# B&R Automation Studio project MotionProyect
Automation Studio 4.11.2.75; Proyecto para realizar las practicas realizada para el curso de motion 27-11-24; technology packages: Acp10Arnc0 5.15.1

## Configuration Demo

CPU 4PPC70.0702-23B, AutomationRuntime F4.92, Build 4.1.2, Safety 0.0, Vc V4.72.5

### Task classes (Cpu.sw)
```
Cyclic#4:
  AxisProgra <- Source.AxisProgram.prg
Libraries: McBase, CoTrace, AsZip, FileIO, runtime, MpAxis, McAxis, MpBase, McAcpAx
```

### Hardware
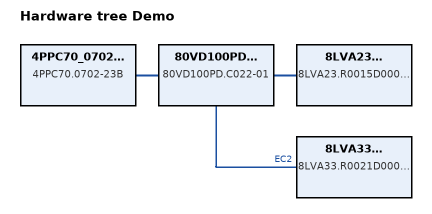
```
4PPC70_0702_23B : 4PPC70.0702-23B v1.5.4.0
  Connector IF2:
    ActivateDevice = 1
    Mode = Manual
    InternetAddress = 192.168.150.95
    SubnetMask = 255.255.255.0
    ActivateSnmp = 2
  ConfigurationID = mappMotion_Demo
  FileDevice1
  FileDeviceName1 = USER
  FileDevicePath1 = USER_PATH
  ActivateOpcUa = 1
  OpcUaInformationModels_PV_Version = 1
  KeyMappingFile = VC\4PPC70_0702_23B.dis
80VD100PD.C022-01 : 80VD100PD.C022-01 v2.5.0.0  [PLK1 -> 4PPC70_0702_23B.IF1 (NodeNumber=2) [Cable Type=PowerlinkCable, Length=10, Version=1.0.0.3]; EC1 -> 8LVA23.R0015D000-0.EC; EC2 -> 8LVA33.R0021D000-0.EC; MT2 -> 8LVA33.R0021D000-0.MT]
  DriveConfiguration/Module:
    McAcoposTypeID = AcoposMicroDConfig
    ActivateACOPOSSimulationOnPLC = 0
  DriveConfiguration/Encoder/EncoderX6A/InterfaceType:
    ResolverPolepairs = 1
  DriveConfiguration/Encoder/EncoderX6B/InterfaceType:
    ResolverPolepairs = 1
  DriveConfiguration/Channel[1]/RealAxis:
    AxisReference = gAxis_1
    MechanicalElementsIsInvisible = 0
  DriveConfiguration/Channel[1]/RealAxis/MechanicalElements/Gearbox:
    InputIsReadOnly = 0
    Input = 1
    OutputIsReadOnly = 0
    Output = 1
  DriveConfiguration/Channel[1]/RealAxis/MechanicalElements/RotaryToLinearTransformation:
    ReferenceDistanceIsReadOnly = 0
    ReferenceDistance = 1
  DriveConfiguration/Channel[1]/RealAxis/Controller:
    ModeIsReadOnly = 0
    Mode = PositionController
  DriveConfiguration/Channel[1]/RealAxis/Controller/Mode/Position:
    ProportionalGain = 50.0
    IntegrationTime = 0.0
    PredictionTime = 0.0004
    TotalDelayTime = 0.0004
  DriveConfiguration/Channel[1]/RealAxis/Controller/Mode/Speed:
    ProportionalGainIsReadOnly = 0
    ProportionalGain = 2.0
    IntegrationTimeIsReadOnly = 0
    IntegrationTime = 0.0
    FilterTimeIsReadOnly = 0
    FilterTime = 0.0
  DriveConfiguration/Channel[1]/RealAxis/Controller/Mode/LoopFilters:
    LoopFilterXIsReadOnly = 0
    LoopFilter1 = NotUsed
    LoopFilter2 = NotUsed
    LoopFilter3 = NotUsed
  DriveConfiguration/Channel[1]/RealAxis/Homing:
    ModeIsReadOnly = 0
    Mode = Direct
  DriveConfiguration/Channel[1]/RealAxis/Homing/Mode:
    Position = 0.0
    ReferencePulse = NotUsed
  DriveConfiguration/Channel[1]/RealAxis/Homing:
    RestorePositionVariable = 
  DriveConfiguration/Channel[1]/RealAxis/StopReaction:
    QuickstopIsReadOnly = 0
    Quickstop = DecelerationLimit
    DriveErrorIsReadOnly = 0
    DriveError = DecelerationLimit
  DriveConfiguration/Channel[1]/RealAxis/MovementErrorLimits:
    PositionError = 1.0
    VelocityErrorMonitoring = Automatic1
  DriveConfiguration/Channel[1]/RealAxis:
    JerkFilterIsReadOnly = 0
    JerkFilter = NotUsed
  DriveConfiguration/Channel[1]/RealAxis/DigitalInputs/HomingSwitch:
    SourceIsReadOnly = 0
    Source = NotUsed
    Level = High
  DriveConfiguration/Channel[1]/RealAxis/DigitalInputs/PositiveLimitSwitch:
    SourceIsReadOnly = 0
    Source = NotUsed
    Level = High
  DriveConfiguration/Channel[1]/RealAxis/DigitalInputs/NegativeLimitSwitch:
    SourceIsReadOnly = 0
    Source = NotUsed
    Level = High
  DriveConfiguration/Channel[1]/RealAxis/DigitalInputs/Trigger1:
    Source = X2Trigger1
    Level = High
  DriveConfiguration/Channel[1]/RealAxis/DigitalInputs/Trigger2:
    Source = X2Trigger2
    Level = High
  DriveConfiguration/Channel[1]/RealAxis/DigitalInputs/Quickstop:
    Input = Trigger2
  DriveConfiguration/Channel[1]/RealAxis/Simulation:
    SimulationModeOnPLC = SetValueGeneration
    SimulationModeOnACOPOS = NotUsed
  DriveConfiguration/Channel[2]/RealAxis:
    AxisReference = gAxis_2
    MechanicalElementsIsInvisible = 0
  DriveConfiguration/Channel[2]/RealAxis/MechanicalElements/Gearbox:
    InputIsReadOnly = 0
    Input = 1
    OutputIsReadOnly = 0
    Output = 1
  DriveConfiguration/Channel[2]/RealAxis/MechanicalElements/RotaryToLinearTransformation:
    ReferenceDistanceIsReadOnly = 0
    ReferenceDistance = 1
  DriveConfiguration/Channel[2]/RealAxis/Controller:
    ModeIsReadOnly = 0
    Mode = PositionController
  DriveConfiguration/Channel[2]/RealAxis/Controller/Mode/Position:
    ProportionalGain = 50.0
    IntegrationTime = 0.0
    PredictionTime = 0.0004
    TotalDelayTime = 0.0004
  DriveConfiguration/Channel[2]/RealAxis/Controller/Mode/Speed:
    ProportionalGainIsReadOnly = 0
    ProportionalGain = 2.0
    IntegrationTimeIsReadOnly = 0
    IntegrationTime = 0.0
    FilterTimeIsReadOnly = 0
    FilterTime = 0.0
  DriveConfiguration/Channel[2]/RealAxis/Controller/Mode/LoopFilters:
    LoopFilterXIsReadOnly = 0
    LoopFilter1 = NotUsed
    LoopFilter2 = NotUsed
    LoopFilter3 = NotUsed
  DriveConfiguration/Channel[2]/RealAxis/Homing:
    ModeIsReadOnly = 0
    Mode = Direct
  DriveConfiguration/Channel[2]/RealAxis/Homing/Mode:
    Position = 0.0
    ReferencePulse = NotUsed
  DriveConfiguration/Channel[2]/RealAxis/Homing:
    RestorePositionVariable = 
  DriveConfiguration/Channel[2]/RealAxis/StopReaction:
    QuickstopIsReadOnly = 0
    Quickstop = DecelerationLimit
    DriveErrorIsReadOnly = 0
    DriveError = DecelerationLimit
  DriveConfiguration/Channel[2]/RealAxis/MovementErrorLimits:
    PositionError = 1.0
    VelocityErrorMonitoring = Automatic1
  DriveConfiguration/Channel[2]/RealAxis:
    JerkFilterIsReadOnly = 0
    JerkFilter = NotUsed
  DriveConfiguration/Channel[2]/RealAxis/DigitalInputs/HomingSwitch:
    SourceIsReadOnly = 0
    Source = NotUsed
    Level = High
  DriveConfiguration/Channel[2]/RealAxis/DigitalInputs/PositiveLimitSwitch:
    SourceIsReadOnly = 0
    Source = NotUsed
    Level = High
  DriveConfiguration/Channel[2]/RealAxis/DigitalInputs/NegativeLimitSwitch:
    SourceIsReadOnly = 0
    Source = NotUsed
    Level = High
  DriveConfiguration/Channel[2]/RealAxis/DigitalInputs/Trigger1:
    Source = X2Trigger1
    Level = High
  DriveConfiguration/Channel[2]/RealAxis/DigitalInputs/Trigger2:
    Source = X2Trigger2
    Level = High
  DriveConfiguration/Channel[2]/RealAxis/DigitalInputs/Quickstop:
    Input = Trigger2
  DriveConfiguration/Channel[2]/RealAxis/Simulation:
    SimulationModeOnPLC = SetValueGeneration
    SimulationModeOnACOPOS = NotUsed
8LVA23.R0015D000-0 : 8LVA23.R0015D000-0 v2.2.0.3  [EC -> 80VD100PD.C022-01.EC1; MT -> 80VD100PD.C022-01.MT1]
  M1/MotorParameters:
    MOTOR_AMB_TEMP_RATED = 40
8LVA33.R0021D000-0 : 8LVA33.R0021D000-0 v2.2.0.3  [EC -> 80VD100PD.C022-01.EC2; MT -> 80VD100PD.C022-01.MT2]
  M1/MotorParameters:
    MOTOR_AMB_TEMP_RATED = 40
```

### IoMap.iom - 4PPC70_0702_23B/IoMap.iom
```iecst
VAR_CONFIG
	::AxisSequence.io.di_PowerMotors AT %IX."4XP0043.00-00W".DigitalInput01;
	::AxisSequence.io.di_StartSequence AT %IX."4XP0043.00-00W".DigitalInput02;
	::AxisSequence.io.di_StopSequence AT %IX."4XP0043.00-00W".DigitalInput03;
END_VAR
```

### Acp10cfg.ncc - 4PPC70_0702_23B/Motion/Acp10cfg.ncc
```
NcConfiguration (Version=5.15.1, NcSwId=Acp10)
  ACP10CF1_typ:
    cnt_nettrc_rec_drive = 1500
    bufsize_trace_upload = 1200
    tc_nc_man_task = Cyclic #1
    glob_pv_as_ncobject = Yes
    ncsys_dl_broadcast = Yes
    ncsys_dl_acp_reset = Yes
    safemc_log_err_to_ax = Yes
    network_init:
      ncsw_init_execute = Yes
      automatic_execute = No
      node_nr_warning = Yes
      net_err_before_ncact = Yes
    nettrc:
      enter_parsecrec = Yes
      enter_ncaction = Yes
      save_ring_startidx = Yes
    cam_prof_download:
      cam_dat_dl_parallel = No
      tc_cam_dl_parallel = Task class for NC Manager task
    plk_if[0]:
      if_name = IF1
      tc_CycDat_PLCopen = Task class for NC Manager task
      mc_broadcast_extdat = No
```

### Acp10map.ncm - 4PPC70_0702_23B/Motion/Acp10map.ncm
```
NcMapping (NcSwId=Acp10, DisabledNodesAreHidden=False)
  NcObject gAxis02 (ModuleId=80VD100PD.C022-01, Type=ncAXIS, Channel=2, AcoposSimulation=Off, InitParameter=gAxis02i, AcoposParameter=gAxis02a, AdditionalData=PLCopen_ModPos="36000,100" , Disabled=FALSE, ModuleDisabled=FALSE)
  NcObject gAxis01 (ModuleId=80VD100PD.C022-01, Type=ncAXIS, Channel=1, AcoposSimulation=Off, InitParameter=gAxis01i, AcoposParameter=gAxis01a, AdditionalData=PLCopen_ModPos="36000,100" , Disabled=FALSE, ModuleDisabled=FALSE)
  NcObject 80VD100PD.C022-01_ncV_AXIS2 (ModuleId=80VD100PD.C022-01, Type=ncV_AXIS, Channel=2, Disabled=TRUE, ModuleDisabled=FALSE)
  NcObject 80VD100PD.C022-01_ncV_AXIS1 (ModuleId=80VD100PD.C022-01, Type=ncV_AXIS, Channel=1, Disabled=TRUE, ModuleDisabled=FALSE)
```

### Axis1.axis - 4PPC70_0702_23B/mappMotion/Axis1.axis
```
Element gAxis_1 (Type=axis)
  BaseTypeIsReadOnly = 0
  BaseType = RotaryPeriodic
    MeasurementUnitIsReadOnly = 0
    MeasurementUnit = 17476
    MeasurementResolutionIsReadOnly = 0
    MeasurementResolution = 0.01
    CountDirectionIsReadOnly = 0
    CountDirection = Standard
    PeriodSettings:
      Period = 360.0
  MovementLimitsIsReadOnly = 0
  MovementLimits = Internal
    Position:
      LowerLimitMin = -1.79769313486231E308
      UpperLimitMax = 1.79769313486231E308
      LowerLimit = -1000.0
      UpperLimit = 1000.0
    VelocityIsReadOnly = 0
    Velocity:
      VelocityMax = 3.4E38
      Velocity = 1000
    AccelerationIsReadOnly = 0
    Acceleration:
      AccelerationMax = 3.4E38
      Acceleration = 1000
    DecelerationIsReadOnly = 0
    Deceleration:
      DecelerationMax = 3.4E38
      Deceleration = 1000
  Alarms = None
```

### Axis2.axis - 4PPC70_0702_23B/mappMotion/Axis2.axis
```
Element gAxis_2 (Type=axis)
  BaseTypeIsReadOnly = 0
  BaseType = RotaryPeriodic
    MeasurementUnitIsReadOnly = 0
    MeasurementUnit = 17476
    MeasurementResolutionIsReadOnly = 0
    MeasurementResolution = 0.01
    CountDirectionIsReadOnly = 0
    CountDirection = Standard
    PeriodSettings:
      Period = 360.0
  MovementLimitsIsReadOnly = 0
  MovementLimits = Internal
    Position:
      LowerLimitMin = -1.79769313486231E308
      UpperLimitMax = 1.79769313486231E308
      LowerLimit = -1000.0
      UpperLimit = 1000.0
    VelocityIsReadOnly = 0
    Velocity:
      VelocityMax = 3.4E38
      Velocity = 1400
    AccelerationIsReadOnly = 0
    Acceleration:
      AccelerationMax = 3.4E38
      Acceleration = 1000
    DecelerationIsReadOnly = 0
    Deceleration:
      DecelerationMax = 3.4E38
      Deceleration = 1000
  Alarms = None
```

### CfgAutomat.axisfeature - 4PPC70_0702_23B/mappMotion/CfgAutomat.axisfeature
```
Element Feature_1 (Type=axisfeature)
  Type = CamAutomat
    CamAutomatType = ACOPOS
      CommonParameters:
        Master:
          ValueSource = SetPosition
            AxisReference = gAxis_1
            MaxVelocity = 30
          StartPosition = 0.0
          StartInterval = MasterAxisPeriod
        AdvancedParameters:
          StartStateParameters:
            StartState = 0
            RelMasterStartPos = 0.0
          AdditiveAxes:
            AdditiveMasterValueSource = NotUsed
            AdditiveSlaveValueSource = NotUsed
          MasterStartPositionMode = NotEvaluatedAnew
          ControlSettings:
            CrossLeftBoundary = PositionLimitedHorizontal
            CamChangeImmediately = CurrentMasterMoveDir
          MessageSettings:
            ErrorsInStandby = NoErrorMessages
          TriggerAndLatch:
            Trigger1Delay = 0.0
            Trigger2Delay = 0.0
            SlaveLatchParID = 0
          EventParIDs
          StartIntervals
          Factors:
            SlaveFactorParID = 0
      States:
        State0 = Used
          Events:
            Event[0]:
              Type = StateEnd
              Transition = Immediately
              SynchronousUpdate = NotUsed
              NextState = 1
        State[1]:
          Cam = Predefined
            PredefinedCam = OneToOne
          MasterFactor = 600
          SlaveFactor = 0
          CompensationMode = NoCompensation
          AdvancedParameters:
            RepeatCounterInit = 0
            MasterValueSource = CommonMaster
          Events:
            Event[0]:
              Type = Signal1FromPLC
              Transition = EndOfState
              SynchronousUpdate = NotUsed
              NextState = 2
            Event[1]:
              Type = StateEnd
              Transition = Immediately
              SynchronousUpdate = NotUsed
              NextState = 1
        State[2]:
          Cam = Predefined
            PredefinedCam = ZeroPoint
          MasterFactor = 1
          SlaveFactor = 1
          CompensationMode = DistancesBetweenCams
            MasterDistance = 20
            SlaveDistance = 170
            AdvancedParameters = NotUsed
          AdvancedParameters:
            RepeatCounterInit = 0
            MasterValueSource = CommonMaster
          Events:
            Event[0]:
              Type = StateEnd
              Transition = EndOfState
              SynchronousUpdate = NotUsed
              NextState = 3
        State[3]:
          Cam = Predefined
            PredefinedCam = OneToOne
          MasterFactor = 400
          SlaveFactor = 100
          CompensationMode = NoCompensation
          AdvancedParameters:
            RepeatCounterInit = 0
            MasterValueSource = CommonMaster
          Events:
            Event[0]:
              Type = StateEnd
              Transition = EndOfState
              SynchronousUpdate = NotUsed
              NextState = 4
        State[4]:
          Cam = Predefined
            PredefinedCam = ZeroPoint
          MasterFactor = 1
          SlaveFactor = 1
          CompensationMode = DistancesBetweenCams
            MasterDistance = 20
            SlaveDistance = 180
            AdvancedParameters = NotUsed
          AdvancedParameters:
            RepeatCounterInit = 0
            MasterValueSource = CommonMaster
          Events:
            Event[0]:
              Type = StateEnd
              Transition = EndOfState
              SynchronousUpdate = NotUsed
              NextState = 1
            Event[1]:
              Type = Signal1FromPLC
              Transition = EndOfState
              SynchronousUpdate = NotUsed
              NextState = 2
```

## Logical view

Binary libraries used (declarations not repeated): operator, runtime, astime, AsIecCon, McBase 5.20.2, CoTrace, AsZip, FileIO, MpAxis 5.20.2, McAxis 5.20.2, MpBase, McAcpAx 5.20.2

### Global.typ - Global data types
```iecst
TYPE
	AxisSequence_typ : 	STRUCT
		cmd : AxisSequence_cmd_typ;
		status : AxisSequence_status_typ;
		io : AxisSequence_io_typ;
		state : AxisSequence_enum;
		couplingParam : MpAxisCouplingParType;
		camSequencer : USINT;
		parameters : ARRAY[1..MAX_AXIS]OF MpAxisBasicParType;
	END_STRUCT;
	AxisSequence_cmd_typ : 	STRUCT
		AutoTune : ARRAY[1..MAX_AXIS]OF BOOL;
		Enable : ARRAY[1..MAX_AXIS]OF BOOL;
		ErrorReset : ARRAY[1..MAX_AXIS]OF BOOL;
		Update : ARRAY[1..MAX_AXIS]OF BOOL;
		Power : ARRAY[1..MAX_AXIS]OF BOOL;
		Home : ARRAY[1..MAX_AXIS]OF BOOL;
		MoveVelocity : ARRAY[1..MAX_AXIS]OF BOOL;
		MoveAbsolute : ARRAY[1..MAX_AXIS]OF BOOL;
		MoveAdditive : ARRAY[1..MAX_AXIS]OF BOOL;
		Stop : ARRAY[1..MAX_AXIS]OF BOOL;
		JogPositive : ARRAY[1..MAX_AXIS]OF BOOL;
		JogNegative : ARRAY[1..MAX_AXIS]OF BOOL;
	END_STRUCT;
	AxisSequence_status_typ : 	STRUCT
		PowerMotors : BOOL;
		StartSequence : BOOL;
		StopSequence : BOOL;
		Active : ARRAY[1..MAX_AXIS]OF BOOL;
		Error : ARRAY[1..MAX_AXIS]OF BOOL;
		StatusID : ARRAY[1..MAX_AXIS]OF DINT;
		UpdateDone : ARRAY[1..MAX_AXIS]OF BOOL;
		Position : ARRAY[1..MAX_AXIS]OF LREAL;
		Velocity : ARRAY[1..MAX_AXIS]OF REAL;
		CommandBusy : ARRAY[1..MAX_AXIS]OF BOOL;
		CommandAborted : ARRAY[1..MAX_AXIS]OF BOOL;
		PowerOn : ARRAY[1..MAX_AXIS]OF BOOL;
		IsHomed : ARRAY[1..MAX_AXIS]OF BOOL;
		InVelocity : ARRAY[1..MAX_AXIS]OF BOOL;
		InPosition : ARRAY[1..MAX_AXIS]OF BOOL;
		MoveActive : ARRAY[1..MAX_AXIS]OF BOOL;
		MoveDone : ARRAY[1..MAX_AXIS]OF BOOL;
		Info : ARRAY[1..MAX_AXIS]OF MpAxisBasicInfoType;
	END_STRUCT;
	AxisSequence_io_typ : 	STRUCT
		di_PowerMotors : BOOL;
		di_StartSequence : BOOL;
		di_StopSequence : BOOL;
	END_STRUCT;
	AxisSequence_enum :
		(
		DISABLED := 0,
		WAIT := 5,
		STEP_1 := 10,
		STEP_2 := 20,
		STEP_3 := 30,
		STEP_4 := 40,
		STEP_5 := 50,
		STEP_6 := 60,
		STEP_7 := 70,
		STEP_8 := 80,
		ERROR := 100
		);
END_TYPE
```

### Constans.var
```iecst
VAR CONSTANT
	MAX_AXIS : USINT := 2;
END_VAR
```

### Global.var - Global variables
```iecst
VAR
	MpAxisBasic_0 : ARRAY[1..MAX_AXIS] OF MpAxisBasic;
	AxisParameters : ARRAY[1..MAX_AXIS] OF MpAxisBasicParType;
	AxisInfo : ARRAY[1..MAX_AXIS] OF MpAxisBasicInfoType;
END_VAR
```


### Program Logical/Source/AxisProgram (IEC)

#### Main.st - Init, cyclic, exit code
```iecst
PROGRAM _INIT
	(* INIT AXIS *)
	FOR i:= 1 TO MAX_AXIS DO

		MpAxisBasic_0[i].Enable	:= TRUE;

		AxisParameters[i].Position		:= 100;
		AxisParameters[i].Velocity		:= 10.0;
		AxisParameters[i].Acceleration	:= 50.0;
		AxisParameters[i].Deceleration	:= 50.0;

	END_FOR;

END_PROGRAM

PROGRAM _CYCLIC

	(* CYCLIC AXIS *)
	MpAxisBasic_0[1].MpLink		:= ADR(gAxis_1);
	MpAxisBasic_0[1].Parameters	:= ADR(AxisParameters[1]);
	AxisInfo[1]					:= MpAxisBasic_0[1].Info;
	MpAxisBasic_0[1]();

	MpAxisBasic_0[2].MpLink		:= ADR(gAxis_2);
	MpAxisBasic_0[2].Parameters	:= ADR(AxisParameters[2]);
	AxisInfo[2]					:= MpAxisBasic_0[2].Info;
	MpAxisBasic_0[2]();

END_PROGRAM

PROGRAM _EXIT

	(* EXIT AXIS *)
	FOR i:= 1 TO MAX_AXIS DO
		MpAxisBasic_0[1].Enable	:= FALSE;
	END_FOR;

END_PROGRAM
```

#### Types.typ - Local data types
```iecst
TYPE
	AxisSequence_typ : 	STRUCT
		cmd : AxisSequence_cmd_typ;
		status : AxisSequence_status_typ;
		io : AxisSequence_io_typ;
		state : AxisSequence_enum;
	END_STRUCT;
	AxisSequence_cmd_typ : 	STRUCT
		Enable : ARRAY[1..MAX_AXIS]OF BOOL;
		ErrorReset : ARRAY[1..MAX_AXIS]OF BOOL;
		Update : ARRAY[1..MAX_AXIS]OF BOOL;
		Power : ARRAY[1..MAX_AXIS]OF BOOL;
		Home : ARRAY[1..MAX_AXIS]OF BOOL;
		MoveVelocity : ARRAY[1..MAX_AXIS]OF BOOL;
		MoveAbsolute : ARRAY[1..MAX_AXIS]OF BOOL;
		Stop : ARRAY[1..MAX_AXIS]OF BOOL;
		JogPositive : ARRAY[1..MAX_AXIS]OF BOOL;
		JogNegative : ARRAY[1..MAX_AXIS]OF BOOL;
	END_STRUCT;
	AxisSequence_status_typ : 	STRUCT
		PowerMotors : BOOL;
		StartSequence : BOOL;
		StopSequence : BOOL;
		Active : ARRAY[1..MAX_AXIS]OF BOOL;
		Error : ARRAY[1..MAX_AXIS]OF BOOL;
		StatusID : ARRAY[1..MAX_AXIS]OF BOOL;
		UpdateDone : ARRAY[1..MAX_AXIS]OF BOOL;
		Position : ARRAY[1..MAX_AXIS]OF BOOL;
		Velocity : ARRAY[1..MAX_AXIS]OF BOOL;
		CommandBusy : ARRAY[1..MAX_AXIS]OF BOOL;
		CommandAborted : ARRAY[1..MAX_AXIS]OF BOOL;
		PowerOn : ARRAY[1..MAX_AXIS]OF BOOL;
		IsHomed : ARRAY[1..MAX_AXIS]OF BOOL;
		InVelocity : ARRAY[1..MAX_AXIS]OF BOOL;
		InPosition : ARRAY[1..MAX_AXIS]OF BOOL;
		MoveActive : ARRAY[1..MAX_AXIS]OF BOOL;
		MoveDone : ARRAY[1..MAX_AXIS]OF BOOL;
	END_STRUCT;
	AxisSequence_io_typ : 	STRUCT
	END_STRUCT;
	AxisSequence_enum :
		(
		WAIT := 0,
		STEP_1 := 10,
		STEP_2 := 20,
		STEP_3 := 30,
		STEP_4 := 40,
		STEP_5 := 50,
		STEP_6 := 60,
		STEP_7 := 70,
		STEP_8 := 80,
		ERROR := 100
		);
END_TYPE
```

#### Variables.var
```iecst
VAR
	AxisSequence : AxisSequence_typ;
	i : USINT;
END_VAR
```

#### Sequences.st
```iecst
ACTION AutoSequence180Action:

END_ACTION
```

### Program Logical/Source/AxisCtrl (IEC)

#### Main.st - Init, cyclic, exit code
```iecst
PROGRAM _INIT
	(* INIT AXIS *)
	FOR i:= 1 TO MAX_AXIS DO

		MpAxisBasic_0[i].Enable	:= TRUE;

		AxisSequence.parameters[i].Position		:= 100;
		AxisSequence.parameters[i].Velocity		:= 10.0;
		AxisSequence.parameters[i].Acceleration	:= 50.0;
		AxisSequence.parameters[i].Deceleration	:= 50.0;

	END_FOR;
	(* CYCLIC AXIS *)
	MpAxisBasic_0[1].MpLink		:= ADR(gAxis_1);
	MpAxisBasic_0[1].Parameters	:= ADR(AxisSequence.parameters[1]);
	MpAxisBasic_0[1]();

	MpAxisBasic_0[2].MpLink		:= ADR(gAxis_2);
	MpAxisBasic_0[2].Parameters	:= ADR(AxisSequence.parameters[2]);
	MpAxisBasic_0[2]();

//	AxisSequence.couplingParam.Gear.RatioDenominator 	:= 3600;
//	AxisSequence.couplingParam.Gear.RatioNumerator		:= -3600;
//	MpAxisCoupling_0.MpLinkMaster	:= ADR(gAxis_1);
//	MpAxisCoupling_0.MpLink 		:= ADR(gAxis_2);
//	MpAxisCoupling_0.Parameters		:= ADR(AxisSequence.couplingParam);
	//	MpAxisCoupling_0.Enable			:= TRUE;

	MpAxisCamSequencer_0.MpLinkMaster 	:= ADR(gAxis_1);
	MpAxisCamSequencer_0.MpLink			:= ADR(gAxis_2);
	MpAxisCamSequencer_0.Parameters		:= ADR(CamSequencerParam);
	MpAxisCamSequencer_0.Enable 		:= TRUE;
	CamSequencerParam.CamSequence.Data.DataAddress	:= ADR (CamAutomatParam);
	MpAxisCamSequencer_0();

END_PROGRAM

PROGRAM _CYCLIC
	MpAxisCamSequencer_0.Signal1		:= AxisSequence.io.di_PowerMotors;
	IF EnableSequence THEN
		TapSequencerAction;
	END_IF;

	MpAxisBasic_0[1]();
	MpAxisBasic_0[2]();

	MpAxisCamSequencer_0();
	//MpAxisCoupling_0();
	(* Axis actions *)
	//AxisCtrlCmdAction;

//	/////////// PHYSICAL INPUTS ///////////
//	AxisSequence.status.PowerMotors		:= AxisSequence.io.di_PowerMotors;
//	AxisSequence.status.StartSequence	:= AxisSequence.io.di_StartSequence;
//	AxisSequence.status.StopSequence	:= AxisSequence.io.di_StopSequence;
//
//
//
//	//Timer poweroff condition
//	TON_TurnOffMotors.PT	:= T#2s;
//
//	IF (AxisSequence.status.StopSequence)  THEN
//		TON_TurnOffMotors.IN	:= TRUE;
//	ELSE
//		TON_TurnOffMotors.IN := FALSE;
//	END_IF;
//
//
//
//	FOR i:= 1 TO MAX_AXIS DO
//
//		IF (AxisSequence.state <> STEP_4) AND NOT (AxisSequence.state = STEP_1) THEN
//			AxisSequence.parameters[i].Distance		:= 180;
//			AxisSequence.parameters[i].Velocity		:= 100;
//			AxisSequence.parameters[i].Acceleration := 1000;
//			AxisSequence.parameters[i].Deceleration := 1000;
//			AxisSequence.parameters[i].Direction := mcDIR_POSITIVE;
//		ELSIF (AxisSequence.state = STEP_4) THEN
//			AxisSequence.parameters[i].Distance		:= -540;
//			AxisSequence.parameters[i].Velocity		:= 100;
//			AxisSequence.parameters[i].Acceleration := 1000;
//			AxisSequence.parameters[i].Deceleration := 1000;
//			AxisSequence.parameters[i].Direction 	:= mcDIR_NEGATIVE;
//
//		END_IF;
//
//		//PowerOn condition
//		IF EDGEPOS(AxisSequence.status.PowerMotors)  THEN
//			MpAxisBasic_0[1].Power	:= TRUE;
//			MpAxisBasic_0[2].Power	:= TRUE;
//		END_IF;
//
//		//Stop condition
//		IF AxisSequence.status.StopSequence OR ResetSequence THEN
//			MpAxisBasic_0[i].Home			:= FALSE;
//			MpAxisBasic_0[i].MoveAbsolute	:= FALSE;
//			MpAxisBasic_0[i].MoveAdditive	:= FALSE;
//			MpAxisBasic_0[i].MoveVelocity	:= FALSE;
//			ResetSequence	:= FALSE;
//			//MpAxisBasic_0[i].Stop			:= TRUE;
//			AxisSequence.state	 			:= STEP_1;
//		ELSE
//			//MpAxisBasic_0[i].Stop 		:= FALSE;
//			MpAxisBasic_0[i].ErrorReset	:= FALSE;
//		END_IF;
//
//		//PowerOff condition
//		IF TON_TurnOffMotors.Q  	THEN
//			MpAxisBasic_0[i].Power			:= FALSE;
//			MpAxisBasic_0[i].Home			:= FALSE;
//			MpAxisBasic_0[i].MoveAbsolute	:= FALSE;
//			MpAxisBasic_0[i].MoveAdditive	:= FALSE;
//			MpAxisBasic_0[i].MoveVelocity	:= FALSE;
//			MpAxisBasic_0[i].Stop			:= TRUE;
//			MpAxisBasic_0[i].ErrorReset		:= TRUE;
//			ResetSequence	:= FALSE;
//			AxisSequence.state	 			:= WAIT;
//		END_IF;
//
//
//		//Error condition
//		IF 	MpAxisBasic_0[i].Error THEN
//			AxisSequence.state	:= ERROR;
//		END_IF;
//
//
//
//
//		CASE AxisSequence.state OF
//
//			DISABLED:
//
//				IF 	MpAxisBasic_0[1].Info.ReadyToPowerOn AND (MpAxisBasic_0[2].Info.ReadyToPowerOn) THEN
//					AxisSequence.state	:= WAIT;
//				ELSE
//
//				END_IF;
//
//			WAIT:
//
//				MpAxisBasic_0[i].Stop:= FALSE;
//
//				IF	MpAxisBasic_0[i].Power AND MpAxisBasic_0[i].PowerOn THEN
//					AxisSequence.state	:= STEP_1;
//				END_IF;
//
//			STEP_1:
//
//
//
//				IF (AxisSequence.status.StartSequence) AND (OldStartSequence <> AxisSequence.status.StartSequence) THEN
//					AxisSequence.parameters[1].Homing.Position 	:= 30;
//					AxisSequence.parameters[2].Homing.Position	:= 200;
//					AxisSequence.parameters[1].Homing.Mode 	:= mcHOMING_DIRECT ;
//					AxisSequence.parameters[2].Homing.Mode 	:= mcHOMING_DIRECT ;
//					MpAxisBasic_0[1].Home	:= TRUE;
//					MpAxisBasic_0[2].Home	:= TRUE;
//					PermissionToHome		:= TRUE;
//				END_IF;
//
//				IF (MpAxisBasic_0[1].IsHomed AND MpAxisBasic_0[2].IsHomed) AND (MpAxisBasic_0[1].Position = 30)
//					AND MpAxisBasic_0[2].Position = 200 AND PermissionToHome AND (CountSequence = 0) THEN
//
//					MpAxisBasic_0[1].Home	:= FALSE;
//					MpAxisBasic_0[2].Home	:= FALSE;
//					PermissionToHome		:= FALSE;
//					PermissionToStart		:= TRUE;
//
//				END_IF;
//
//				IF PermissionToStart THEN
//					AxisSequence.parameters[1].Position	:= 0;
//					AxisSequence.parameters[2].Position	:= 0;
//					AxisSequence.parameters[1].Direction := mcDIR_SHORTEST_WAY;
//					AxisSequence.parameters[2].Direction := mcDIR_SHORTEST_WAY;
//
//					MpAxisBasic_0[1].MoveAbsolute	:= TRUE;
//					MpAxisBasic_0[2].MoveAbsolute	:= TRUE;
//				END_IF;
//
//				IF MpAxisBasic_0[1].InPosition AND MpAxisBasic_0[1].MoveDone THEN
//					MpAxisBasic_0[1].MoveAbsolute	:= FALSE;
//					FinishSequence[1]				:= TRUE;
//				END_IF;
//
//				IF MpAxisBasic_0[2].InPosition AND MpAxisBasic_0[2].MoveDone THEN
//					MpAxisBasic_0[2].MoveAbsolute	:= FALSE;
//					FinishSequence[2]				:= TRUE;
//				END_IF;
//
//				IF FinishSequence[1] AND FinishSequence[2] THEN
//					FinishSequence[1]		:= FALSE;
//					FinishSequence[2]		:= FALSE;
//					PermissionToStart		:= FALSE;
//					CountSequence			:= 1;
//					AxisSequence.state		:= STEP_2;
//				END_IF;
//
//			STEP_2: //+180° Axis 1
//
//				IF (CountSequence <7) THEN
//					MpAxisBasic_0[1].MoveAdditive	:= TRUE;
//					IF MpAxisBasic_0[1].InPosition AND (MpAxisBasic_0[1].MoveDone) THEN
//						MpAxisBasic_0[1].MoveAdditive	:= FALSE;
//						CountSequence 					:= CountSequence + 1;
//						AxisSequence.state				:= STEP_3;
//					END_IF;
//				END_IF;
//
//				IF (CountSequence = 7) THEN
//					AxisSequence.state	:= STEP_4;
//				END_IF;
//
//			STEP_3: //+180 Axis 2
//
//				IF (CountSequence <7) THEN
//					MpAxisBasic_0[2].MoveAdditive := TRUE;
//					IF MpAxisBasic_0[2].InPosition AND (MpAxisBasic_0[2].MoveDone) THEN
//						MpAxisBasic_0[2].MoveAdditive	:= FALSE;
//						CountSequence 					:= CountSequence + 1;
//						AxisSequence.state				:= STEP_2;
//					END_IF;
//				END_IF;
//
//			STEP_4:
//
//				MpAxisBasic_0[i].MoveAdditive := TRUE;
//
//				IF MpAxisBasic_0[1].InPosition AND MpAxisBasic_0[1].MoveDone THEN
//					MpAxisBasic_0[1].MoveAdditive	:= FALSE;
//					FinishSequence[1]				:= TRUE;
//				END_IF;
//
//				IF MpAxisBasic_0[2].InPosition AND MpAxisBasic_0[2].MoveDone THEN
//					MpAxisBasic_0[2].MoveAdditive	:= FALSE;
//					FinishSequence[2]				:= TRUE;
//				END_IF;
//
//				IF FinishSequence[1] AND FinishSequence[2] THEN
//					FinishSequence[1]		:= FALSE;
//					FinishSequence[2]		:= FALSE;
//					ResetSequence			:= TRUE;
//					CountSequence			:= 0;
//					AxisSequence.state		:= STEP_1;
//				END_IF;
//
//
//			ERROR:
//
//				MpAxisBasic_0[i].MoveAdditive	:= FALSE;
//				IF NOT(MpAxisBasic_0[1].Error) AND NOT(MpAxisBasic_0[2].Error)THEN
//					AxisSequence.state	:= WAIT;
//				END_IF;
//
//
//		END_CASE;
//
//
//		MpAxisBasic_0[i]();
//	END_FOR;
//
//
//	//Old variables
//	OldStartSequence := AxisSequence.status.StartSequence;
//
//	//Call Functions blocks
//	//AxisCtrlStatusAction;
//	TON_TurnOffMotors();
//

END_PROGRAM

PROGRAM _EXIT

	(* EXIT AXIS *)
	FOR i:= 1 TO MAX_AXIS DO
		MpAxisBasic_0[i].Enable	:= FALSE;
	END_FOR;

END_PROGRAM
```

#### Variables.var
```iecst
VAR
	MpAxisBasic_0 : ARRAY[1..MAX_AXIS] OF MpAxisBasic;
	i : USINT;
	PermissionToStart : BOOL;
	TON_TurnOffMotors : TON;
	OldStartSequence : BOOL;
	FinishSequence : ARRAY[1..MAX_AXIS] OF BOOL;
	CountSequence : USINT;
	HomePosition : ARRAY[1..MAX_AXIS] OF LREAL;
	PermissionToHome : BOOL;
	ResetSequence : BOOL;
	MpAxisCoupling_0 : MpAxisCoupling;
	MpAxisCamSequencer_0 : MpAxisCamSequencer;
	CamSequencerParam : MpAxisCamSequencerParType;
	CamAutomatParam : McAcpAxCamAutParType;
	EnableSequence : BOOL;
END_VAR
```

#### TapSequencerAction.st
```iecst
ACTION TapSequencerAction:
//no detecta botellas

	EnableSequence	:= FALSE;

	CamAutomatParam.State[0].CamID						:= 16#FFFF;
	CamAutomatParam.State[0].Event[0].Type				:= mcEVENT_STATE_END;
	CamAutomatParam.State[0].Event[0].Transition		:= mcEVENT_IMMEDIATELY;
	CamAutomatParam.State[0].Event[0].NextState			:= 1;

	CamAutomatParam.State[1].CamID										:= 16#FFFF;
	CamAutomatParam.State[1].MasterFactor								:= 1080;
	CamAutomatParam.State[1].SlaveFactor								:= 0;
	CamAutomatParam.State[1].CompensationMode							:= mcCOMP_OFF;
	CamAutomatParam.State[1].CompensationParameters.MasterCompDistance	:= 0;
	CamAutomatParam.State[1].CompensationParameters.SlaveCompDistance	:= 0;
	CamAutomatParam.State[1].Event[0].Type				:= mcEVENT_SIGNAL1;
	CamAutomatParam.State[1].Event[0].Transition		:= mcEVENT_END_OF_STATE;
	CamAutomatParam.State[1].Event[0].NextState			:= 2;

	CamAutomatParam.State[1].Event[1].Type				:= mcEVENT_STATE_END;
	CamAutomatParam.State[1].Event[1].Transition		:= mcEVENT_IMMEDIATELY;
	CamAutomatParam.State[1].Event[1].NextState			:= 1;

	CamAutomatParam.State[2].CamID										:= 16#FFFE;
	CamAutomatParam.State[2].MasterFactor								:= 1;
	CamAutomatParam.State[2].SlaveFactor								:= 1;
	CamAutomatParam.State[2].CompensationMode							:= mcCOMP_BETWEEN_CAMS;
	CamAutomatParam.State[2].CompensationParameters.MasterCompDistance	:= 108;
	CamAutomatParam.State[2].CompensationParameters.SlaveCompDistance	:= -146;
	CamAutomatParam.State[2].Event[0].Type				:= mcEVENT_STATE_END;
	CamAutomatParam.State[2].Event[0].Transition		:= mcEVENT_END_OF_STATE;
	CamAutomatParam.State[2].Event[0].NextState			:= 3;

	CamAutomatParam.State[3].CamID										:= 16#FFFF;
	CamAutomatParam.State[3].MasterFactor								:= 720;
	CamAutomatParam.State[3].SlaveFactor								:= -720;
	CamAutomatParam.State[3].CompensationMode							:= mcCOMP_OFF;
	CamAutomatParam.State[3].CompensationParameters.MasterCompDistance	:= 0;
	CamAutomatParam.State[3].CompensationParameters.SlaveCompDistance	:= 0;
	CamAutomatParam.State[3].Event[0].Type					:= mcEVENT_STATE_END;
	CamAutomatParam.State[3].Event[0].Transition			:= mcEVENT_END_OF_STATE;
	CamAutomatParam.State[3].Event[0].NextState				:= 4;

	CamAutomatParam.State[4].CamID										:= 16#FFFE;
	CamAutomatParam.State[4].MasterFactor								:= 1;
	CamAutomatParam.State[4].SlaveFactor								:= 1;
	CamAutomatParam.State[4].CompensationMode							:= mcCOMP_BETWEEN_CAMS;
	CamAutomatParam.State[4].CompensationParameters.MasterCompDistance	:= 108;
	CamAutomatParam.State[4].CompensationParameters.SlaveCompDistance	:= -142;
	CamAutomatParam.State[4].Event[0].Type					:= mcEVENT_SIGNAL1;
	CamAutomatParam.State[4].Event[0].Transition			:= mcEVENT_END_OF_STATE;
	CamAutomatParam.State[4].Event[0].NextState				:= 2;
	CamAutomatParam.State[4].Event[1].Type					:= mcEVENT_STATE_END;
	CamAutomatParam.State[4].Event[1].Transition			:= mcEVENT_END_OF_STATE;
	CamAutomatParam.State[4].Event[1].NextState				:= 1;

END_ACTION
```

#### MpAxisActions.st - not listed in the package file held
```iecst
ACTION AxisCtrlStatusAction:

	FOR i:=1 TO MAX_AXIS DO

		AxisSequence.status.Active[i]			:= MpAxisBasic_0[i].Active;
		AxisSequence.status.CommandAborted[i]	:= MpAxisBasic_0[i].CommandAborted;
		AxisSequence.status.CommandBusy[i]		:= MpAxisBasic_0[i].CommandBusy;
		AxisSequence.status.Error[i]			:= MpAxisBasic_0[i].Error;
		AxisSequence.status.InPosition[i]		:= MpAxisBasic_0[i].InPosition;
		AxisSequence.status.InVelocity[i]		:= MpAxisBasic_0[i].InVelocity;
		AxisSequence.status.IsHomed[i]			:= MpAxisBasic_0[i].IsHomed;
		AxisSequence.status.MoveActive[i]		:= MpAxisBasic_0[i].MoveActive;
		AxisSequence.status.MoveDone[i]			:= MpAxisBasic_0[i].MoveDone;
		AxisSequence.status.Position[i]			:= MpAxisBasic_0[i].Position;
		AxisSequence.status.PowerOn[i]			:= MpAxisBasic_0[i].PowerOn;
		AxisSequence.status.StatusID[i]			:= MpAxisBasic_0[i].StatusID;
		AxisSequence.status.UpdateDone[i]		:= MpAxisBasic_0[i].UpdateDone;
		AxisSequence.status.Velocity[i]			:= MpAxisBasic_0[i].Velocity;
		AxisSequence.status.Info[i]				:= MpAxisBasic_0[i].Info;

	END_FOR;

END_ACTION
```

### Program Logical/Source/AxisSequence

#### Variables.var
```iecst
VAR
	TON_TurnOffMotors : TON;
	i : USINT;
END_VAR
```

#### Main.st
```iecst
PROGRAM _INIT
	(* Insert code here *)

END_PROGRAM

PROGRAM _CYCLIC

	/////////// PHYSICAL INPUTS ///////////
	AxisSequence.status.PowerMotors		:= AxisSequence.io.di_PowerMotors;
	AxisSequence.status.StartSequence	:= AxisSequence.io.di_StartSequence;
	AxisSequence.status.StopSequence	:= AxisSequence.io.di_StopSequence;

	//Timer poweroff condition
	TON_TurnOffMotors.PT	:= T#2s;

	IF (AxisSequence.status.StopSequence)  THEN
		TON_TurnOffMotors.IN	:= TRUE;
	ELSE
		TON_TurnOffMotors.IN := FALSE;
	END_IF;

	FOR i:= 1 TO MAX_AXIS DO

		IF AxisSequence.state <> (STEP_8) THEN
			AxisSequence.parameters[i].Distance		:= 180;
			AxisSequence.parameters[i].Velocity		:= 1000;
			AxisSequence.parameters[i].Acceleration := 7200;
			AxisSequence.parameters[i].Deceleration := 7200;
		ELSIF AxisSequence.state = (STEP_8) THEN
			AxisSequence.parameters[i].Distance		:= -540;
			AxisSequence.parameters[i].Velocity		:= 1500;
			AxisSequence.parameters[i].Acceleration := 7200;
			AxisSequence.parameters[i].Deceleration := 7200;
		END_IF;

		//PowerOn condition
		IF EDGEPOS(AxisSequence.status.PowerMotors)  THEN
			AxisSequence.cmd.Power[i]	:= TRUE;
		END_IF;

		//Stop condition
		IF AxisSequence.status.StopSequence THEN
			AxisSequence.cmd.Home[i]			:= FALSE;
			AxisSequence.cmd.MoveAbsolute[i]	:= FALSE;
			AxisSequence.cmd.MoveAdditive[i]	:= FALSE;
			AxisSequence.cmd.MoveVelocity[i]	:= FALSE;
			AxisSequence.cmd.Stop[i]			:= TRUE;
		ELSE
			AxisSequence.cmd.Stop[i] := FALSE;
		END_IF;

		//PowerOff condition
		IF TON_TurnOffMotors.Q  	THEN
			AxisSequence.cmd.Power[i]			:= FALSE;
			AxisSequence.cmd.Home[i]			:= FALSE;
			AxisSequence.cmd.MoveAbsolute[i]	:= FALSE;
			AxisSequence.cmd.MoveAdditive[i]	:= FALSE;
			AxisSequence.cmd.MoveVelocity[i]	:= FALSE;
			AxisSequence.cmd.Stop[i]			:= TRUE;
			AxisSequence.state	 				:= WAIT;
		END_IF;

		//Error condition
		IF AxisSequence.status.Error[i] THEN
			AxisSequence.state	:= ERROR;
		END_IF;

		CASE AxisSequence.state OF

			WAIT:

				IF	AxisSequence.cmd.Power[i] AND AxisSequence.status.PowerOn[i] THEN
					AxisSequence.state	:= STEP_1;
				END_IF;

			STEP_1:

				IF	EDGEPOS(AxisSequence.status.StartSequence) THEN
				//	AxisSequence.cmd.MoveAbsolute[i]			:= TRUE;
					AxisSequence.cmd.Home[i]					:= TRUE;
				END_IF;

				IF (*(AxisSequence.status.InPosition[1]) AND (AxisSequence.status.MoveDone[1]) AND
				   (AxisSequence.status.InPosition[2]) AND (AxisSequence.status.MoveDone[2]) THEN *)
					(AxisSequence.status.IsHomed[1] AND AxisSequence.status.IsHomed[2]) THEN

					AxisSequence.cmd.Home[i]					:= FALSE;
					AxisSequence.cmd.MoveAdditive[1]			:= TRUE;

				END_IF;

				IF AxisSequence.status.InPosition[1] AND (AxisSequence.status.MoveDone[1]) THEN
					//AutoSequence.cmd.homeMode		:= mcHOME_DEFAULT;
					AxisSequence.cmd.MoveAdditive[1]	:= FALSE;
					//AutoSequence.cmd.home			:= FALSE;
					AxisSequence.state					:= STEP_2;
				END_IF;

			STEP_2: //+180° Axis 2

					AxisSequence.cmd.MoveAdditive[2] := TRUE;

					IF AxisSequence.status.InPosition[2] AND (AxisSequence.status.MoveDone[2]) THEN
						AxisSequence.cmd.MoveAdditive[2]	:= FALSE;
						AxisSequence.state					:= STEP_3;
					END_IF;

			STEP_3: //+180 Axis 1
					AxisSequence.cmd.MoveAdditive[1] := TRUE;

					IF AxisSequence.status.InPosition[1] AND (AxisSequence.status.MoveDone[1]) THEN
						AxisSequence.cmd.MoveAdditive[1]	:= FALSE;
						AxisSequence.state					:= STEP_4;
					END_IF;

			STEP_4: //+180 Axis 2

					AxisSequence.cmd.MoveAdditive[2] := TRUE;

					IF AxisSequence.status.InPosition[2] AND (AxisSequence.status.MoveDone[2]) THEN
						AxisSequence.cmd.MoveAdditive[2]	:= FALSE;
						AxisSequence.state					:= STEP_5;
					END_IF;

			STEP_5:	//+180 Axis 1

					AxisSequence.cmd.MoveAdditive[1] := TRUE;

					IF AxisSequence.status.InPosition[1] AND (AxisSequence.status.MoveDone[1]) THEN
						AxisSequence.cmd.MoveAdditive[1]	:= FALSE;
						AxisSequence.state					:= STEP_6;
					END_IF;

			STEP_6: //+180 Axis 2

					AxisSequence.cmd.MoveAdditive[2] := TRUE;

					IF AxisSequence.status.InPosition[2] AND (AxisSequence.status.MoveDone[2]) THEN
						AxisSequence.cmd.MoveAdditive[2]	:= FALSE;
						AxisSequence.state					:= STEP_7;
					END_IF;

			STEP_7: //+180 Axis 1

					AxisSequence.cmd.MoveAdditive[2] := TRUE;

					IF AxisSequence.status.InPosition[2] AND (AxisSequence.status.MoveDone[2]) THEN
						AxisSequence.cmd.MoveAdditive[2]	:= FALSE;
						AxisSequence.state					:= STEP_8;
					END_IF;

			STEP_8:

					AxisSequence.cmd.MoveAdditive[i] := TRUE;

					IF AxisSequence.status.InPosition[1] AND AxisSequence.status.InPosition[2] THEN
						AxisSequence.cmd.MoveAdditive[2]	:= FALSE;
						AxisSequence.state					:= STEP_8;
					END_IF;

			ERROR:

				AxisSequence.cmd.MoveAdditive[i]	:= FALSE;
				IF NOT(AxisSequence.status.Error[1]) AND NOT(AxisSequence.status.Error[1])THEN
						AxisSequence.state	:= WAIT;
				END_IF;

			END_CASE;

	END_FOR;

	//Call Functions blocks
	TON_TurnOffMotors();

END_PROGRAM

PROGRAM _EXIT
	(* Insert code here *)

END_PROGRAM
```

### Constants.var - not listed in the package file held
```iecst
VAR CONSTANT
	AXIS_SHIFT_FORWARD : USINT := 0;
	AXIS_SHIFT_REVERSE : USINT := 1;
END_VAR
```

### Package Logical/Sources/MotionObjects/gAxis01obj - gAxis01obj

### gAxis01i.ax
```
InitParameter (Version=5.15.1, NcSwId=Acp10)
  ACP10AXIS_typ:
    dig_in:
      level:
        reference = ncACTIV_HI
        pos_hw_end = ncACTIV_HI
        neg_hw_end = ncACTIV_HI
        trigger1 = ncACTIV_HI
        trigger2 = ncACTIV_HI
    encoder_if:
      parameter:
        count_dir = ncSTANDARD
        scaling:
          load:
            units = 36000
            rev_motor = 1
    limit:
      parameter:
        v_pos = 198000.0
        v_neg = 198000.0
        a1_pos = 1980000.0
        a2_pos = 1980000.0
        a1_neg = 1980000.0
        a2_neg = 1980000.0
        t_jolt = 0
        t_in_pos = 0
        pos_sw_end = 2000000000
        neg_sw_end = -2000000000
        ds_warning = 500
        ds_stop = 1000
        a_stop = 1.0e30
        dv_stop = 0
        dv_stop_mode = ncOFF
    controller:
      mode = ncPOSITION
      position:
        kv = 50
        tn = 0
        t_predict = 0.0004
        t_total = 0.0004
        p_max = 1.0e30
        i_max = 0
      speed:
        kv = 2.0
        tn = 0
        t_filter = 0.0
        isq_filter1:
          type = ncOFF
          a0 = 0.0
          a1 = 0.0
          b0 = 0.0
          b1 = 0.0
          b2 = 0.0
          c0_par_id = 0
          c1_par_id = 0
        isq_filter2:
          type = ncOFF
          a0 = 0.0
          a1 = 0.0
          b0 = 0.0
          b1 = 0.0
          b2 = 0.0
          c0_par_id = 0
          c1_par_id = 0
        isq_filter3:
          type = ncOFF
          a0 = 0.0
          a1 = 0.0
          b0 = 0.0
          b1 = 0.0
          b2 = 0.0
          c0_par_id = 0
          c1_par_id = 0
      uf:
        type = ncLINEAR + ncCORRECTION
        auto_config = ncMOTOR_PAR
        u0 = 0
        un = 0
        fn = 50.0
        k_f_slip = 0
      ff:
        mode = ncSTANDARD
        torque_load = 0.0
        torque_pos = 0.0
        torque_neg = 0.0
        kv_torque = 0.0
        inertia = 0.0
        t_filter_a = 0.0
      fb:
        mode = ncSTANDARD
        speed_mix_ratio = 0.0
        speed_kv = 2.0
      model:
        mass1:
          inertia = 0
          viscous_friction = 0
        mass2:
          inertia = 0
          viscous_friction = 0
          stiffness = 0
          damping = 0
    move:
      stop:
        parameter[0]:
          decel_ramp = ncA_LIMIT
          controller = ncON
        parameter[1]:
          decel_ramp = ncA_LIMIT
          controller = ncON
        parameter[2]:
          decel_ramp = ncA_LIMIT
          controller = ncON
        parameter[3]:
          decel_ramp = ncA_LIMIT
          controller = ncON
        quickstop:
          decel_ramp = ncA_LIMIT
          t_jolt = 0
        drive_error:
          decel_ramp = ncA_LIMIT
      homing:
        parameter:
          s = 0
          v_switch = 5000
          v_trigger = 500
          a = 50000
          mode = ncDIRECT
          edge_sw = ncPOSITIVE
          start_dir = ncPOSITIVE
          trigg_dir = ncPOSITIVE
          ref_pulse = ncOFF
          fix_dir = ncOFF
          tr_s_block = 0
          torque_lim = 0
          ds_block = 0
          ds_stop = 0
      basis:
        parameter:
          v_pos = 5000
          v_neg = 5000
          a1_pos = 50000
          a2_pos = 50000
          a1_neg = 50000
          a2_neg = 50000
    message:
      text:
        parameter:
          format = ncBREAK
          columns = 80
          data_modul = acp10etxen
```

### Package Logical/Sources/MotionObjects/gAxis02obj - gAxis02obj

### gAxis02i.ax
```
InitParameter (Version=5.15.1, NcSwId=Acp10)
  ACP10AXIS_typ:
    dig_in:
      level:
        reference = ncACTIV_HI
        pos_hw_end = ncACTIV_HI
        neg_hw_end = ncACTIV_HI
        trigger1 = ncACTIV_HI
        trigger2 = ncACTIV_HI
    encoder_if:
      parameter:
        count_dir = ncSTANDARD
        scaling:
          load:
            units = 36000
            rev_motor = 1
    limit:
      parameter:
        v_pos = 366000.0
        v_neg = 366000.0
        a1_pos = 3660000.0
        a2_pos = 3660000.0
        a1_neg = 3660000.0
        a2_neg = 3660000.0
        t_jolt = 0
        t_in_pos = 0
        pos_sw_end = 2000000000
        neg_sw_end = -2000000000
        ds_warning = 500
        ds_stop = 1000
        a_stop = 1.0e30
        dv_stop = 0
        dv_stop_mode = ncOFF
    controller:
      mode = ncPOSITION
      position:
        kv = 50
        tn = 0
        t_predict = 0.0004
        t_total = 0.0004
        p_max = 1.0e30
        i_max = 0
      speed:
        kv = 2.0
        tn = 0
        t_filter = 0.0
        isq_filter1:
          type = ncOFF
          a0 = 0.0
          a1 = 0.0
          b0 = 0.0
          b1 = 0.0
          b2 = 0.0
          c0_par_id = 0
          c1_par_id = 0
        isq_filter2:
          type = ncOFF
          a0 = 0.0
          a1 = 0.0
          b0 = 0.0
          b1 = 0.0
          b2 = 0.0
          c0_par_id = 0
          c1_par_id = 0
        isq_filter3:
          type = ncOFF
          a0 = 0.0
          a1 = 0.0
          b0 = 0.0
          b1 = 0.0
          b2 = 0.0
          c0_par_id = 0
          c1_par_id = 0
      uf:
        type = ncLINEAR + ncCORRECTION
        auto_config = ncMOTOR_PAR
        u0 = 0
        un = 0
        fn = 50.0
        k_f_slip = 0
      ff:
        mode = ncSTANDARD
        torque_load = 0.0
        torque_pos = 0.0
        torque_neg = 0.0
        kv_torque = 0.0
        inertia = 0.0
        t_filter_a = 0.0
      fb:
        mode = ncSTANDARD
        speed_mix_ratio = 0.0
        speed_kv = 2.0
      model:
        mass1:
          inertia = 0
          viscous_friction = 0
        mass2:
          inertia = 0
          viscous_friction = 0
          stiffness = 0
          damping = 0
    move:
      stop:
        parameter[0]:
          decel_ramp = ncA_LIMIT
          controller = ncON
        parameter[1]:
          decel_ramp = ncA_LIMIT
          controller = ncON
        parameter[2]:
          decel_ramp = ncA_LIMIT
          controller = ncON
        parameter[3]:
          decel_ramp = ncA_LIMIT
          controller = ncON
        quickstop:
          decel_ramp = ncA_LIMIT
          t_jolt = 0
        drive_error:
          decel_ramp = ncA_LIMIT
      homing:
        parameter:
          s = 0
          v_switch = 5000
          v_trigger = 500
          a = 50000
          mode = ncDIRECT
          edge_sw = ncPOSITIVE
          start_dir = ncPOSITIVE
          trigg_dir = ncPOSITIVE
          ref_pulse = ncOFF
          fix_dir = ncOFF
          tr_s_block = 0
          torque_lim = 0
          ds_block = 0
          ds_stop = 0
      basis:
        parameter:
          v_pos = 5000
          v_neg = 5000
          a1_pos = 50000
          a2_pos = 50000
          a1_neg = 50000
          a2_neg = 50000
    message:
      text:
        parameter:
          format = ncBREAK
          columns = 80
          data_modul = acp10etxen
```

### Data object Logical/Sources/MotionObjects/acp10etxen (Ett)

- acp10etxen.ett (not shown)

### Variables.var - Local variables
```iecst
VAR
	AxisSecuence : USINT;
	CountCycle : USINT;
	TON_TurnOffMotors : TON;
	PWM_Active : MTBasicsPWM;
	i : USINT;
	CountManualSequence : USINT;
	OldStartMotor : BOOL;
END_VAR
```

### Program Logical/Sources/MotionControl/AutoSequence (IEC)

#### Main.st - Init, cyclic, exit code
```iecst
PROGRAM _INIT
	(* Insert code here *)
	 AutoSequence.par.speedMovement := 100;
END_PROGRAM

PROGRAM _CYCLIC
	(*///////////////////// PHYSICAL INPUTS /////////////////////*)
	AutoSequence.status.powerMotors	:= AutoSequence.io.di_PowerMotors;
	AutoSequence.status.startMotors	:= AutoSequence.io.di_StartSequence;
	AutoSequence.status.stopMotor	:= AutoSequence.io.di_StopSequence;

	TON_TurnOffMotors.PT	:= T#2s;

	IF NOT(AutoSequence.cmd.AutoSequenceDisabled) THEN
		IF EDGEPOS(AutoSequence.status.powerMotors)  THEN
			AutoSequence.status.doPowerMotorsOff		:= FALSE;
			AutoSequence.status.doPowerMotorsON			:= TRUE;
			AutoSequence.cmd.powerMotor	:= TRUE;
		END_IF;
	END_IF
	IF (AutoSequence.status.powerMotors)  THEN
		TON_TurnOffMotors.IN	:= TRUE;
	ELSE
		TON_TurnOffMotors.IN := FALSE;
	END_IF;

	IF AutoSequence.status.stopMotor THEN
		AutoSequence.status.doStopCycleActive := TRUE;
	ELSE
		AutoSequence.status.doStopCycleActive := FALSE;
	END_IF;

	IF TON_TurnOffMotors.Q  OR (AutoSequence.status.stopMotor)	THEN
		AutoSequence.cmd.powerMotor					:= FALSE;
		AutoSequence.cmd.moveRelative[1]			:= FALSE;
		AutoSequence.cmd.moveRelative[2]			:= FALSE;
		AutoSequence.status.homePositionOk[1]		:= FALSE;
		AutoSequence.status.homePositionOk[2]		:= FALSE;
		AutoSequence.status.doPowerMotorsOff		:= TRUE;
		AutoSequence.status.doPowerMotorsON			:= FALSE;
		AutoSequence.status.doStartCycleInactive	:= TRUE;
		AutoSequence.status.doStartCycleActive		:= FALSE;
		AutoSequence.state	 := WAIT;
	END_IF;

	IF AutoSequence.state <> (STEP_8) THEN
		AutoSequence.par.speedMovement;
		AutoSequence.par.acceleration		:= 7200;
		AutoSequence.par.deceleration		:= 7200;
	ELSIF AutoSequence.state = (STEP_8) THEN
		AutoSequence.par.speedMovement;
		AutoSequence.par.acceleration		:= 7200;
		AutoSequence.par.deceleration		:= 7200;
	ELSIF AutoSequence.cmd.AutoSequenceDisabled THEN
		AutoSequence.par.speedMovement;
		AutoSequence.par.acceleration;
		AutoSequence.par.deceleration;
	END_IF

	IF AutoSequence.status.errorActive[1] OR AutoSequence.status.errorActive[2] THEN
		AutoSequence.state	:= ERROR;
	END_IF;

	IF EDGEPOS (AutoSequence.cmd.AutoSequenceDisabled) THEN
		AutoSequence.cmd.powerMotor			:= FALSE;
		AutoSequence.cmd.moveRelative[1]	:= FALSE;
		AutoSequence.cmd.moveRelative[2]	:= FALSE;
		AutoSequence.cmd.home				:= FALSE;
		AutoSequence.par.homeMode			:= mcHOME_DEFAULT;
		AutoSequence.state	:= MANUAL;
	END_IF;

	CASE AutoSequence.state OF

		WAIT:

			IF	AutoSequence.cmd.powerMotor THEN
				AutoSequence.state							:= STEP_1;
			END_IF;

		STEP_1:

			IF	EDGEPOS(AutoSequence.status.startMotors) THEN
				AutoSequence.cmd.startMotor					:= TRUE;
				AutoSequence.status.doStartCycleActive		:= TRUE;
				AutoSequence.status.doStartCycleInactive	:= FALSE;
				AutoSequence.par.position[1];
				AutoSequence.par.position[2];
				AutoSequence.par.direction[1]				:= AXIS_SHIFT_FORWARD;
				AutoSequence.par.direction[2]				:= AXIS_SHIFT_REVERSE;
				AutoSequence.cmd.moveAbsolute[1]			:= TRUE;
				AutoSequence.cmd.moveAbsolute[2]			:= TRUE;
				//AutoSequence.cmd.homeMode				:= mcHOME_ABSOLUTE;
				(*AutoSequence.cmd.home					:= TRUE;*)
			END_IF;

			IF AutoSequence.status.moveAbsoluteDone[1] THEN
				AutoSequence.cmd.moveAbsolute[1]		:= FALSE;
				AutoSequence.status.homePositionOk[1]	:= TRUE;
			END_IF;
			IF AutoSequence.status.moveAbsoluteDone[2] THEN
				AutoSequence.cmd.moveAbsolute[1]		:= FALSE;
				AutoSequence.status.homePositionOk[2] 	:= TRUE;
			END_IF;

			IF AutoSequence.status.homePositionOk[1] AND AutoSequence.status.homePositionOk[2] AND (AutoSequence.cmd.startMotor) THEN
				AutoSequence.cmd.startMotor			:= FALSE;
				//AutoSequence.cmd.homeMode		:= mcHOME_DEFAULT;
				AutoSequence.status.homePositionOk[1]	:= FALSE;
				AutoSequence.status.homePositionOk[2]	:= FALSE;
				AutoSequence.cmd.moveAbsolute[1]		:= FALSE;
				AutoSequence.cmd.moveAbsolute[2]		:= FALSE;
				//AutoSequence.cmd.home			:= FALSE;
				AutoSequence.state					:= STEP_2;
			END_IF;

		STEP_2: //+180° Axis 1

			AutoSequence.par.distance[1]		:= 180;
			AutoSequence.par.direction[1]		:= AXIS_SHIFT_FORWARD;
			IF NOT (AutoSequence.status.stopMotor) THEN
				AutoSequence.cmd.moveRelative[1]	:= TRUE;
			ELSE
				AutoSequence.cmd.moveRelative[1]	:= FALSE;
			END_IF;

			IF AutoSequence.status.MoveAdditiveDone[1] THEN
				AutoSequence.cmd.moveRelative[1]	:= FALSE;
				AutoSequence.state					:= STEP_3;
			END_IF;

		STEP_3: //+180 Axis 2
			AutoSequence.par.distance[2]		:= 180;
			AutoSequence.cmd.moveRelative[2]	:= TRUE;
			AutoSequence.par.direction[2]		:= AXIS_SHIFT_FORWARD;
			IF  (AutoSequence.status.MoveAdditiveDone[2]) THEN
				AutoSequence.cmd.moveRelative[2]	:= FALSE;
				AutoSequence.state					:= STEP_4;
			END_IF;

		STEP_4: //+180 Axis 1
			AutoSequence.par.distance[1]			:= 180;
			AutoSequence.par.direction[1]			:= AXIS_SHIFT_FORWARD;
			IF NOT (AutoSequence.status.stopMotor) THEN
				AutoSequence.cmd.moveRelative[1]	:= TRUE;
			ELSE
				AutoSequence.cmd.moveRelative[1]	:= FALSE;
			END_IF;

			IF AutoSequence.status.MoveAdditiveDone[1] THEN
				AutoSequence.cmd.moveRelative[1]	:= FALSE;
				AutoSequence.state					:= STEP_5;
			END_IF;

		STEP_5:	//+180 Axis 2

			AutoSequence.par.distance[2]		:= 180;
			AutoSequence.cmd.moveRelative[2]	:= TRUE;
			AutoSequence.par.direction[1]		:= AXIS_SHIFT_FORWARD;
			IF (AutoSequence.status.MoveAdditiveDone[2]) THEN
				AutoSequence.cmd.moveRelative[2]	:= FALSE;
				AutoSequence.state					:= STEP_6;
			END_IF;

		STEP_6: //+180 Axis 1
			AutoSequence.par.distance[1]		:= 180;
			AutoSequence.cmd.moveRelative[1]	:= TRUE;
			AutoSequence.par.direction[1]		:= AXIS_SHIFT_FORWARD;

			IF AutoSequence.status.MoveAdditiveDone[1] THEN
				AutoSequence.cmd.moveRelative[1]	:= FALSE;
				AutoSequence.state				:= STEP_7;
			END_IF;

		STEP_7: //+180 Axis 2
			AutoSequence.par.distance[2]		:= 180;
			AutoSequence.cmd.moveRelative[2]	:= TRUE;
			AutoSequence.par.direction[1]		:= AXIS_SHIFT_FORWARD;

			IF  (AutoSequence.status.MoveAdditiveDone[2]) THEN
				AutoSequence.cmd.moveRelative[2]	:= FALSE;
				AutoSequence.cmd.moveRelative[1]	:= TRUE;
				AutoSequence.cmd.moveRelative[2]	:= TRUE;
				AutoSequence.state				:= STEP_8;
			END_IF;

		STEP_8:
			AutoSequence.par.distance[1]		:= -540;
			AutoSequence.par.distance[2]		:= -540;

			AutoSequence.par.direction[1]				:= AXIS_SHIFT_REVERSE;
			AutoSequence.par.direction[2]				:= AXIS_SHIFT_REVERSE;
			IF ( AutoSequence.status.MoveAdditiveDone[1])  THEN
				AutoSequence.cmd.moveRelative[1]		:= FALSE;
				AutoSequence.status.finalPosition[1]	:= TRUE;
			END_IF;

			IF ( AutoSequence.status.MoveAdditiveDone[2])  THEN
				AutoSequence.cmd.moveRelative[2]		:= FALSE;
				AutoSequence.status.finalPosition[2]	:= TRUE;
			END_IF;

			IF AutoSequence.status.finalPosition[1] AND AutoSequence.status.finalPosition[2] THEN
				AutoSequence.cmd.powerMotor				:= FALSE;
				AutoSequence.status.doStartCycleActive	:= FALSE;
				AutoSequence.status.finalPosition[1]	:= FALSE;
				AutoSequence.status.finalPosition[2]	:= FALSE;
				AutoSequence.state						:= WAIT;
			END_IF;

		ERROR:
			AutoSequence.cmd.moveRelative[1]	:= FALSE;
			AutoSequence.cmd.moveRelative[2]	:= FALSE;
			AutoSequence.status.doErrorActive	:= TRUE;
			AutoSequence.status.doPowerMotorsOff		:= FALSE;
			AutoSequence.status.doPowerMotorsON			:= FALSE;
			AutoSequence.status.doStartCycleInactive	:= FALSE;
			AutoSequence.status.doStartCycleActive		:= FALSE;

			IF NOT(AutoSequence.status.errorActive[1]) AND NOT(AutoSequence.status.errorActive[2])
				AND NOT (AutoSequence.cmd.AutoSequenceDisabled) THEN
				AutoSequence.status.doErrorActive	:= FALSE;
				AutoSequence.state	:= WAIT;
			ELSIF	NOT(AutoSequence.status.errorActive[1]) AND NOT(AutoSequence.status.errorActive[2])
				AND AutoSequence.cmd.AutoSequenceDisabled THEN
				AutoSequence.status.doErrorActive	:= FALSE;
				AutoSequence.state	:= MANUAL;
			END_IF;

		MANUAL:

			IF NOT(AutoSequence.cmd.AutoSequenceDisabled) THEN
				AutoSequence.state	:= WAIT;
			END_IF;

	END_CASE;
	OldStartMotor := AutoSequence.status.startMotors;
	LedSequenceAction;

	PWM_Active();
	TON_TurnOffMotors();

END_PROGRAM

PROGRAM _EXIT
	(* Insert code here *)

END_PROGRAM
```

#### LedSequenceAction.st
```iecst
ACTION LedSequenceAction:

	FOR i:= 1 TO 3 DO
		IF AutoSequence.status.doErrorActive THEN
			AutoSequence.io.do_LedBlue			:= FALSE;
			AutoSequence.io.do_LedGreen[i]		:= FALSE;
			AutoSequence.io.do_LedWhite[i]		:= FALSE;
			AutoSequence.io.do_LedYellow[i]		:= FALSE;
			PWM_Active.Enable					:= TRUE;
			PWM_Active.Period					:= 2;
			PWM_Active.DutyCycle				:= 50;
			AutoSequence.io.do_LedRed[i]		:= PWM_Active.Out;
		ELSE
			AutoSequence.io.do_LedRed[i]		:= FALSE;
			PWM_Active.Enable					:= FALSE;
		END_IF;

		IF AutoSequence.cmd.AutoSequenceDisabled AND CountManualSequence <> 3 THEN
			AutoSequence.io.do_LedBlue			:= FALSE;
			AutoSequence.io.do_LedGreen[i]		:= FALSE;
			AutoSequence.io.do_LedWhite[i]		:= FALSE;
			AutoSequence.io.do_LedRed[i]		:= FALSE;
			PWM_Active.Enable					:= TRUE;
			PWM_Active.Period					:= 2;
			PWM_Active.DutyCycle				:= 50;
			AutoSequence.io.do_LedYellow[i]		:= PWM_Active.Out;
			IF EDGEPOS (PWM_Active.Out) THEN
				CountManualSequence := CountManualSequence + 1;
			END_IF;
		ELSIF AutoSequence.cmd.AutoSequenceDisabled AND (CountManualSequence >= 3) THEN
			PWM_Active.Enable					:= FALSE;
			AutoSequence.io.do_LedYellow[i]		:= TRUE;
		ELSIF NOT(AutoSequence.cmd.AutoSequenceDisabled) AND NOT(AutoSequence.status.doErrorActive) THEN
			AutoSequence.io.do_LedBlue			:= FALSE;
			AutoSequence.io.do_LedGreen[i]		:= FALSE;
			AutoSequence.io.do_LedRed[i]		:= FALSE;
			PWM_Active.Enable					:= FALSE;
			AutoSequence.io.do_LedYellow[i]		:= FALSE;
			CountManualSequence					:= 0;
		END_IF;

	END_FOR;

	IF NOT (AutoSequence.status.doErrorActive) AND NOT(AutoSequence.cmd.AutoSequenceDisabled) THEN

		IF AutoSequence.status.doPowerMotorsOff	 OR (AutoSequence.state = WAIT) THEN
			AutoSequence.io.do_LedGreen[1]	:= FALSE;
			AutoSequence.io.do_LedWhite[1]	:= TRUE;
		ELSIF AutoSequence.status.doPowerMotorsON THEN
			AutoSequence.io.do_LedGreen[1]	:= TRUE;
			AutoSequence.io.do_LedWhite[1]	:= FALSE;
		END_IF

		IF AutoSequence.status.doStartCycleInactive OR (AutoSequence.state = WAIT) THEN
			AutoSequence.io.do_LedWhite[2]	:= TRUE;
			AutoSequence.io.do_LedGreen[2]	:= FALSE;
		ELSIF	AutoSequence.status.doStartCycleActive THEN
			AutoSequence.io.do_LedWhite[2]	:= FALSE;
			AutoSequence.io.do_LedGreen[2]	:= TRUE;
		END_IF;

		IF AutoSequence.status.doStopCycleActive THEN
			AutoSequence.io.do_LedBlue		:= TRUE;
		ELSE
			AutoSequence.io.do_LedBlue		:= FALSE;
		END_IF;
	END_IF;

END_ACTION
```

### Program Logical/Sources/MotionControl/BasicAxis1 (IEC) - Basic logical control

#### basicCyclic.st - cyclic code
```iecst
(********************************************************************
 * COPYRIGHT -- Bernecker + Rainer
 ********************************************************************
 * PROGRAM: Basic
 * File: basicCyclic.st
 * Author: Bernecker + Rainer
 * Created: December 01, 2009
 ********************************************************************
 * Implementation of Program Basic
 ********************************************************************)
PROGRAM _CYCLIC

	Axis1Cmd;
	Axis1Param;
	Axis1CyclicReadAction;

(***************************************************************
        Control Sequence
***************************************************************)
(* status information is read before the step sequencer to attain a shorter reaction time *)
(************************ MC_READSTATUS *************************)
MC_ReadStatus_0.Enable := NOT(MC_ReadStatus_0.Error);
MC_ReadStatus_0.Axis := Axis1Obj;
MC_ReadStatus_0();
BasicControl.AxisState.Disabled             := MC_ReadStatus_0.Disabled;
BasicControl.AxisState.StandStill           := MC_ReadStatus_0.StandStill;
BasicControl.AxisState.Stopping             := MC_ReadStatus_0.Stopping;
BasicControl.AxisState.Homing               := MC_ReadStatus_0.Homing;
BasicControl.AxisState.DiscreteMotion       := MC_ReadStatus_0.DiscreteMotion;
BasicControl.AxisState.ContinuousMotion     := MC_ReadStatus_0.ContinuousMotion;
BasicControl.AxisState.SynchronizedMotion   := MC_ReadStatus_0.SynchronizedMotion;
BasicControl.AxisState.ErrorStop            := MC_ReadStatus_0.Errorstop;

(********************MC_BR_READDRIVESTATUS***********************)
MC_BR_ReadDriveStatus_0.Enable := NOT(MC_BR_ReadDriveStatus_0.Error);
MC_BR_ReadDriveStatus_0.Axis := Axis1Obj;
MC_BR_ReadDriveStatus_0.AdrDriveStatus := ADR(BasicControl.Status.DriveStatus);
MC_BR_ReadDriveStatus_0();

(******************** MC_READACTUALPOSITION *********************)
MC_ReadActualPosition_0.Enable := (NOT(MC_ReadActualPosition_0.Error));
MC_ReadActualPosition_0.Axis := Axis1Obj;
MC_ReadActualPosition_0();
IF(MC_ReadActualPosition_0.Valid = TRUE)THEN
    BasicControl.Status.ActPosition := MC_ReadActualPosition_0.Position;
END_IF

(******************** MC_READACTUALVELOCITY *********************)
MC_ReadActualVelocity_0.Enable := (NOT(MC_ReadActualVelocity_0.Error));
MC_ReadActualVelocity_0.Axis := Axis1Obj;
MC_ReadActualVelocity_0();
IF(MC_ReadActualVelocity_0.Valid = TRUE)THEN
    BasicControl.Status.ActVelocity := MC_ReadActualVelocity_0.Velocity;
END_IF

(************************ MC_READAXISERROR **********************)
MC_ReadAxisError_0.Enable := NOT(MC_ReadAxisError_0.Error);
MC_ReadAxisError_0.Axis := Axis1Obj;
MC_ReadAxisError_0.DataAddress := ADR(BasicControl.Status.ErrorText);
MC_ReadAxisError_0.DataLength := SIZEOF(BasicControl.Status.ErrorText);
MC_ReadAxisError_0.DataObjectName := 'acp10etxen';
MC_ReadAxisError_0();

(**************** CHECK FOR GENERAL AXIS ERROR ******************)
    IF ((MC_ReadAxisError_0.AxisErrorID <> 0) AND (MC_ReadAxisError_0.Valid = TRUE)) THEN
        AxisStep := STATE_ERROR_AXIS;
(***************** CHECK IF POWER SHOULD BE OFF *******************)
    ELSIF ((BasicControl.Command.Power = FALSE) AND (MC_ReadAxisError_0.Valid = TRUE)) THEN
        IF ((MC_ReadStatus_0.Errorstop = TRUE) AND (MC_ReadStatus_0.Valid = TRUE)) THEN
            AxisStep := STATE_ERROR_RESET;
        ELSE
            AxisStep := STATE_WAIT;
        END_IF
    END_IF

(* central monitoring OF stop command attains a shorter reaction TIME in CASE OF emergency stop *)
(******************CHECK FOR STOP COMMAND************************)
    IF (BasicControl.Command.Stop = TRUE) THEN
        IF ((AxisStep >= STATE_HOME) AND (AxisStep <= STATE_ERROR)) THEN
            (* reset all FB execute inputs we use *)
            MC_Home_0.Execute := 0;
            MC_Stop_0.Execute := 0;
            MC_MoveAbsolute_0.Execute := 0;
            MC_MoveAdditive_0.Execute := 0;
            MC_MoveVelocity_0.Execute := 0;
            MC_ReadAxisError_0.Acknowledge := 0;
            MC_Reset_0.Execute := 0;
            MC_Halt_0.Execute := 0;

            (* reset user commands *)
            BasicControl.Command.Halt := 0;
            BasicControl.Command.Home := 0;
            BasicControl.Command.MoveJogPos := 0;
            BasicControl.Command.MoveJogNeg := 0;
            BasicControl.Command.MoveVelocity := 0;
            BasicControl.Command.MoveAbsolute := 0;
            BasicControl.Command.MoveAdditive := 0;
            AxisStep := STATE_STOP;
        END_IF
    END_IF

CASE AxisStep OF

(******************** WAIT *************************)
    STATE_WAIT:  (* STATE: Wait *)
        IF (BasicControl.Command.Power = TRUE) THEN
            AxisStep := STATE_POWER_ON;
        ELSE
            MC_Power_0.Enable := FALSE;
        END_IF

        (* reset all FB execute inputs we use *)
        MC_Home_0.Execute := FALSE;
        MC_Stop_0.Execute := FALSE;
        MC_MoveAbsolute_0.Execute := FALSE;
        MC_MoveAdditive_0.Execute := FALSE;
        MC_MoveVelocity_0.Execute := FALSE;
        MC_Halt_0.Execute := FALSE;
        MC_ReadAxisError_0.Acknowledge := FALSE;
        MC_Reset_0.Execute := FALSE;

        (* reset user commands *)
        BasicControl.Command.Stop := FALSE;
        BasicControl.Command.Halt := FALSE;
        BasicControl.Command.Home := FALSE;
        BasicControl.Command.MoveJogPos := FALSE;
        BasicControl.Command.MoveJogNeg := FALSE;
        BasicControl.Command.MoveVelocity := FALSE;
        BasicControl.Command.MoveAbsolute := FALSE;
        BasicControl.Command.MoveAdditive := FALSE;

        BasicControl.Status.ErrorID := 0;

(******************** POWER ON **********************)
    STATE_POWER_ON:  (* STATE: Power on *)
        MC_Power_0.Enable := TRUE;
        IF (MC_Power_0.Status = TRUE) THEN
            AxisStep := STATE_READY;
        END_IF
        (* if a power error occured go to error state *)
        IF (MC_Power_0.Error = TRUE) THEN
            BasicControl.Status.ErrorID := MC_Power_0.ErrorID;
            AxisStep := STATE_ERROR;
        END_IF

(******************** READY **********************)
    STATE_READY:  (* STATE: Waiting for commands *)
        IF (BasicControl.Command.Home = TRUE)THEN
            BasicControl.Command.Home := FALSE;
            AxisStep := STATE_HOME;

        ELSIF (BasicControl.Command.Stop = TRUE) THEN
            AxisStep := STATE_STOP;

        ELSIF (BasicControl.Command.MoveJogPos = TRUE) THEN
            AxisStep := STATE_JOG_POSITIVE;

        ELSIF (BasicControl.Command.MoveJogNeg = TRUE) THEN
            AxisStep := STATE_JOG_NEGATIVE;

        ELSIF (BasicControl.Command.MoveAbsolute = TRUE) THEN
            BasicControl.Command.MoveAbsolute := FALSE;
            AxisStep := STATE_MOVE_ABSOLUTE;

        ELSIF (BasicControl.Command.MoveAdditive = TRUE) THEN
            BasicControl.Command.MoveAdditive := FALSE;
            AxisStep := STATE_MOVE_ADDITIVE;

        ELSIF (BasicControl.Command.MoveVelocity = TRUE) THEN
            BasicControl.Command.MoveVelocity := FALSE;
            AxisStep := STATE_MOVE_VELOCITY;

        ELSIF (BasicControl.Command.Halt = TRUE) THEN
            BasicControl.Command.Halt := FALSE;
            AxisStep := STATE_HALT;
        END_IF

(******************** HOME **********************)
    STATE_HOME:  (* STATE: start homing process *)
        MC_Home_0.Position := BasicControl.Parameter.HomePosition;
        MC_Home_0.HomingMode := BasicControl.Parameter.HomeMode;
        MC_Home_0.Execute := TRUE;
        IF (MC_Home_0.Done = TRUE) THEN
            MC_Home_0.Execute := FALSE;
            AxisStep := STATE_READY;
        END_IF
        (* if a homing error occured go to error state *)
        IF (MC_Home_0.Error = TRUE) THEN
            MC_Home_0.Execute := FALSE;
            BasicControl.Status.ErrorID := MC_Home_0.ErrorID;
            AxisStep := STATE_ERROR;
        END_IF

(***********************HALT_MOVEMENT***************************)
    STATE_HALT:   (* STATE: Halt movement *)
        MC_Halt_0.Deceleration := BasicControl.Parameter.Deceleration;
        MC_Halt_0.Execute := TRUE;
        IF (MC_Halt_0.Done = TRUE) THEN
            MC_Halt_0.Execute := FALSE;
            AxisStep := STATE_READY;
        END_IF
        (* check if error occured *)
        IF (MC_Halt_0.Error = TRUE) THEN
            BasicControl.Status.ErrorID := MC_Halt_0.ErrorID;
            MC_Halt_0.Execute := FALSE;
            AxisStep := STATE_ERROR;
        END_IF

(*********************** STOP MOVEMENT *************************)
    STATE_STOP:  (* STATE: Stop movement *)
        MC_Stop_0.Deceleration := BasicControl.Parameter.Deceleration;
        MC_Stop_0.Execute := TRUE;
        (* if axis is stopped go to ready state *)
        IF ((MC_Stop_0.Done = TRUE) AND (BasicControl.Command.Stop = FALSE)) THEN
            MC_Stop_0.Execute := FALSE;
            AxisStep := STATE_READY;
        END_IF
        (* check if error occured *)
        IF (MC_Stop_0.Error = TRUE) THEN
            BasicControl.Status.ErrorID := MC_Stop_0.ErrorID;
            MC_Stop_0.Execute := FALSE;
            AxisStep := STATE_ERROR;
        END_IF

(******************** START JOG MOVEMENT POSITVE **********************)
     STATE_JOG_POSITIVE:  (* STATE: Start jog movement in positive direction *)
        MC_MoveVelocity_0.Velocity      := BasicControl.Parameter.JogVelocity;
        MC_MoveVelocity_0.Acceleration  := BasicControl.Parameter.Acceleration;
        MC_MoveVelocity_0.Deceleration  := BasicControl.Parameter.Deceleration;
        MC_MoveVelocity_0.Direction     := mcPOSITIVE_DIR;
        MC_MoveVelocity_0.Execute := TRUE;
        IF (BasicControl.Command.MoveJogPos = FALSE) THEN
            MC_MoveVelocity_0.Execute := FALSE;
            AxisStep := STATE_HALT;
        END_IF
        (* check if error occured *)
        IF (MC_MoveVelocity_0.Error = TRUE) THEN
            BasicControl.Status.ErrorID := MC_MoveVelocity_0.ErrorID;
            MC_MoveVelocity_0.Execute := FALSE;
            AxisStep := STATE_ERROR;
        END_IF

(******************** START JOG MOVEMENT NEGATIVE **********************)
    STATE_JOG_NEGATIVE:  (* STATE: Start jog movement in negative direction *)
        MC_MoveVelocity_0.Velocity      := BasicControl.Parameter.JogVelocity;
        MC_MoveVelocity_0.Acceleration  := BasicControl.Parameter.Acceleration;
        MC_MoveVelocity_0.Deceleration  := BasicControl.Parameter.Deceleration;
        MC_MoveVelocity_0.Direction	    := mcNEGATIVE_DIR;
        MC_MoveVelocity_0.Execute := TRUE;
        IF (BasicControl.Command.MoveJogNeg = FALSE) THEN
            MC_MoveVelocity_0.Execute := FALSE;
            AxisStep := STATE_HALT;
        END_IF
        (* check if error occured *)
        IF (MC_MoveVelocity_0.Error = TRUE) THEN
            BasicControl.Status.ErrorID := MC_MoveVelocity_0.ErrorID;
            MC_MoveVelocity_0.Execute := FALSE;
            AxisStep := STATE_ERROR;
        END_IF

(******************** START ABSOLUTE MOVEMENT **********************)
     STATE_MOVE_ABSOLUTE:  (* STATE: Start absolute movement *)
        MC_MoveAbsolute_0.Position      := BasicControl.Parameter.Position;
        MC_MoveAbsolute_0.Velocity      := BasicControl.Parameter.Velocity;
        MC_MoveAbsolute_0.Acceleration  := BasicControl.Parameter.Acceleration;
        MC_MoveAbsolute_0.Deceleration  := BasicControl.Parameter.Deceleration;
        MC_MoveAbsolute_0.Direction     := BasicControl.Parameter.Direction;
        MC_MoveAbsolute_0.Execute := TRUE;
        (* check if commanded position is reached *)
        IF (BasicControl.Command.Halt) THEN
            BasicControl.Command.Halt := FALSE;
            MC_MoveAbsolute_0.Execute := FALSE;
            AxisStep := STATE_HALT;
        ELSIF (MC_MoveAbsolute_0.Done = TRUE) THEN
            MC_MoveAbsolute_0.Execute := FALSE;
            AxisStep := STATE_READY;
        END_IF
        (* check if error occured *)
        IF (MC_MoveAbsolute_0.Error = TRUE) THEN
            BasicControl.Status.ErrorID := MC_MoveAbsolute_0.ErrorID;
            MC_MoveAbsolute_0.Execute := FALSE;
            AxisStep := STATE_ERROR;
        END_IF

(******************** START ADDITIVE MOVEMENT **********************)
    STATE_MOVE_ADDITIVE:  (* STATE: Start additive movement *)
        MC_MoveAdditive_0.Distance      := BasicControl.Parameter.Distance;
        MC_MoveAdditive_0.Velocity      := BasicControl.Parameter.Velocity;
        MC_MoveAdditive_0.Acceleration  := BasicControl.Parameter.Acceleration;
        MC_MoveAdditive_0.Deceleration  := BasicControl.Parameter.Deceleration;
        MC_MoveAdditive_0.Execute := TRUE;
        (* check if commanded distance is reached *)
        IF (BasicControl.Command.Halt) THEN
            BasicControl.Command.Halt := FALSE;
            MC_MoveAdditive_0.Execute := FALSE;
            AxisStep := STATE_HALT;
        ELSIF (MC_MoveAdditive_0.Done = TRUE) THEN
            MC_MoveAdditive_0.Execute := FALSE;
            AxisStep := STATE_READY;
        END_IF
        (* check if error occured *)
        IF (MC_MoveAdditive_0.Error = TRUE) THEN
            BasicControl.Status.ErrorID := MC_MoveAdditive_0.ErrorID;
            MC_MoveAdditive_0.Execute := FALSE;
            AxisStep := STATE_ERROR;
        END_IF

(******************** START VELOCITY MOVEMENT **********************)
    STATE_MOVE_VELOCITY:  (* STATE: Start velocity movement *)
        MC_MoveVelocity_0.Velocity      := BasicControl.Parameter.Velocity;
        MC_MoveVelocity_0.Acceleration  := BasicControl.Parameter.Acceleration;
        MC_MoveVelocity_0.Deceleration  := BasicControl.Parameter.Deceleration;
        MC_MoveVelocity_0.Direction     := BasicControl.Parameter.Direction;
        MC_MoveVelocity_0.Execute := TRUE;
        (* check if commanded velocity is reached *)
        IF (BasicControl.Command.Halt) THEN
            BasicControl.Command.Halt := FALSE;
            MC_MoveVelocity_0.Execute := FALSE;
            AxisStep := STATE_HALT;
        ELSIF (MC_MoveVelocity_0.InVelocity = TRUE) THEN
            MC_MoveVelocity_0.Execute := FALSE;
            AxisStep := STATE_READY;
        END_IF
        (* check if error occured *)
        IF (MC_MoveVelocity_0.Error = TRUE) THEN
            BasicControl.Status.ErrorID := MC_MoveVelocity_0.ErrorID;
            MC_MoveVelocity_0.Execute := FALSE;
            AxisStep := STATE_ERROR;
        END_IF

(******************** FB-ERROR OCCURED *************************)
    STATE_ERROR:  (* STATE: Error *)
        (* check if FB indicates an axis error *)
        IF (MC_ReadAxisError_0.AxisErrorCount<>0) THEN
            AxisStep := STATE_ERROR_AXIS;
        ELSE
            IF (BasicControl.Command.ErrorAcknowledge = TRUE) THEN
                BasicControl.Command.ErrorAcknowledge := FALSE;
                BasicControl.Status.ErrorID := 0;
                (* reset axis if it is in axis state ErrorStop *)
                IF ((MC_ReadStatus_0.Errorstop = TRUE) AND (MC_ReadStatus_0.Valid = TRUE)) THEN
                    AxisStep := STATE_ERROR_RESET;
                ELSE
                    AxisStep := STATE_WAIT;
                END_IF
            END_IF
        END_IF

(******************** AXIS-ERROR OCCURED *************************)
    STATE_ERROR_AXIS:  (* STATE: Axis Error *)
        IF (MC_ReadAxisError_0.Valid = TRUE) THEN
            IF (MC_ReadAxisError_0.AxisErrorID <> 0) THEN
                BasicControl.Status.ErrorID := MC_ReadAxisError_0.AxisErrorID;
            END_IF
            MC_ReadAxisError_0.Acknowledge := FALSE;
            IF (BasicControl.Command.ErrorAcknowledge = TRUE) THEN
                BasicControl.Command.ErrorAcknowledge := FALSE;
                (* acknowledge axis error *)
                IF (MC_ReadAxisError_0.AxisErrorID <> 0) THEN
                    MC_ReadAxisError_0.Acknowledge := TRUE;
                END_IF
            END_IF
            IF (MC_ReadAxisError_0.AxisErrorCount = 0) THEN
                (* reset axis if it is in axis state ErrorStop *)
                BasicControl.Status.ErrorID := 0;
                IF ((MC_ReadStatus_0.Errorstop = TRUE) AND (MC_ReadStatus_0.Valid = TRUE)) THEN
                    AxisStep := STATE_ERROR_RESET;
                ELSE
                    AxisStep := STATE_WAIT;
                END_IF
            END_IF
        END_IF

(******************** RESET DONE *************************)
    STATE_ERROR_RESET:  (* STATE: Wait for reset done *)
        MC_Reset_0.Execute := TRUE;
        (* reset MC_Power.Enable if this FB is in Error*)
        IF (MC_Power_0.Error = TRUE) THEN
            MC_Power_0.Enable := FALSE;
        END_IF
        IF(MC_Reset_0.Done = TRUE)THEN
            MC_Reset_0.Execute := FALSE;
            AxisStep := STATE_WAIT;
        ELSIF(MC_Reset_0.Error = TRUE) THEN
            MC_Reset_0.Execute := FALSE;
            AxisStep := STATE_ERROR;
        END_IF
(******************** SEQUENCE END *************************)
END_CASE

	AutoSequence.status.actPositon[1]			:= BasicControl.Status.ActPosition;
	AutoSequence.status.homingDone[1]			:= MC_Home_0.Done;
	AutoSequence.status.MoveAdditiveDone[1]		:= MC_MoveAdditive_0.Done;
	AutoSequence.status.moveAbsoluteDone[1]		:= MC_MoveAbsolute_0.Done;

	//ERROR OCCURRED
	IF BasicControl.Status.ErrorID <> 0 THEN
		AutoSequence.status.errorActive[1]	:= TRUE;
	ELSE
		AutoSequence.status.errorActive[1]	:= FALSE;
	END_IF;

(***************************************************************
        Function Block Calls
***************************************************************)

(************************** MC_POWER ****************************)
MC_Power_0.Axis := Axis1Obj;  (* pointer to axis *)
MC_Power_0();

(************************** MC_HOME *****************************)
MC_Home_0.Axis := Axis1Obj;
MC_Home_0();

(********************** MC_MOVEABSOLUTE *************************)
MC_MoveAbsolute_0.Axis := Axis1Obj;
MC_MoveAbsolute_0();

(********************** MC_MOVEADDITIVE *************************)
MC_MoveAdditive_0.Axis := Axis1Obj;
MC_MoveAdditive_0();

(********************** MC_MOVEVELOCITY *************************)
MC_MoveVelocity_0.Axis := Axis1Obj;
MC_MoveVelocity_0();

(************************** MC_STOP *****************************)
MC_Stop_0.Axis := Axis1Obj;
MC_Stop_0();

(***************************MC_HALT******************************)
MC_Halt_0.Axis := Axis1Obj;
MC_Halt_0();

(************************** MC_RESET ****************************)
MC_Reset_0.Axis := Axis1Obj;
MC_Reset_0();

END_PROGRAM
```

#### basicInit.st - init code
```iecst
PROGRAM _INIT

	(* get axis object *)
	Axis1Obj := ADR(gAxis01);

	AxisStep := STATE_WAIT; (* start step *)

	BasicControl.Parameter.Velocity             := 1000;  (*velocity for movement*)
	BasicControl.Parameter.Acceleration         := 5000;  (*acceleration for movement*)
	BasicControl.Parameter.Deceleration         := 5000;  (*deceleration for movement*)
	BasicControl.Parameter.JogVelocity          := 400;   (*velocity for jogging *)

END_PROGRAM
```

#### basic.var - Local variables
```iecst
VAR
	BasicControl : basic_typ; (*control structure*)
	MC_Home_0 : MC_Home; (*Function Block*)
	MC_MoveAbsolute_0 : MC_MoveAbsolute; (*Function Block*)
	MC_MoveAdditive_0 : MC_MoveAdditive; (*Function Block*)
	MC_MoveVelocity_0 : MC_MoveVelocity; (*Function Block*)
	MC_Power_0 : MC_Power; (*Function Block*)
	MC_ReadActualPosition_0 : MC_ReadActualPosition; (*Function Block *)
	MC_ReadActualVelocity_0 : MC_ReadActualVelocity; (*Function Block*)
	MC_ReadAxisError_0 : MC_ReadAxisError; (*Function Block*)
	MC_ReadStatus_0 : MC_ReadStatus; (*Function Block*)
	MC_Reset_0 : MC_Reset; (*Function Block*)
	MC_Stop_0 : MC_Stop; (*Function Block*)
	MC_BR_ReadDriveStatus_0 : MC_BR_ReadDriveStatus; (*Function Block*)
	MC_Halt_0 : MC_Halt; (*Function Block*)
	Axis1Obj : UDINT; (*axis reference*)
	AxisStep : UINT; (*current step in the step sequence*)
END_VAR
VAR CONSTANT
	STATE_READY : USINT := 10; (*constant for a waiting step*)
	STATE_POWER_ON : USINT := 1; (*constant for the step in which the controller is switched on*)
	STATE_MOVE_VELOCITY : USINT := 16; (*constant for the step in which a movement with defiened velocity is started*)
	STATE_MOVE_ABSOLUTE : USINT := 14; (*constant for the step in which a movement to defiened position is started*)
	STATE_WAIT : USINT := 0; (*constant for a waiting step*)
	STATE_STOP : USINT := 11; (*constant for the step in which movements are stopped*)
	STATE_MOVE_ADDITIVE : USINT := 15; (*constant for the step in which a movement with defiened distance is started*)
	STATE_HOME : USINT := 2; (*constant for the step in which the axis is homed*)
	STATE_ERROR_RESET : USINT := 102; (*constant for the step in which the errors are reset*)
	STATE_ERROR_AXIS : USINT := 100; (*constant for the axis error step*)
	STATE_ERROR : USINT := 101; (*constant for the error step*)
	STATE_JOG_POSITIVE : USINT := 12; (*constant for the step in which a positive jogging movement is executed*)
	STATE_JOG_NEGATIVE : USINT := 13; (*constant for the step in which a negative jogging movement is executed*)
	STATE_HALT : USINT := 17; (*constant for the step in which movements are stopped*)
END_VAR
VAR
	MC_BR_CyclicRead_0 : MC_BR_CyclicRead;
	MC_BR_CyclicRead_1 : MC_BR_CyclicRead;
	MC_BR_CyclicRead_2 : MC_BR_CyclicRead;
	Axis1MotorTorque : REAL;
	Axis1SensorTemp : REAL;
	Axis1EncoderPosition : DINT;
END_VAR
```

#### BasicAxis1Action.st
```iecst
ACTION Axis1CyclicReadAction:

	MC_BR_CyclicRead_0.Axis			:= ADR(gAxis01);
	MC_BR_CyclicRead_0.Enable		:= TRUE;
	MC_BR_CyclicRead_0.ParID		:= ACP10PAR_TEMP_MOTOR; //Temperature sensor: Temperature
	MC_BR_CyclicRead_0.DataAddress	:= ADR(Axis1SensorTemp);
	MC_BR_CyclicRead_0.DataType		:= ncPAR_TYP_REAL;
	MC_BR_CyclicRead_0.Mode			:= mcEVERY_RECORD;
	MC_BR_CyclicRead_0();

	MC_BR_CyclicRead_1.Axis			:= ADR(gAxis01);
	MC_BR_CyclicRead_1.Enable		:= TRUE;
	MC_BR_CyclicRead_1.ParID		:= ACP10PAR_TORQUE_ACT;
	MC_BR_CyclicRead_1.DataAddress	:= ADR(Axis1MotorTorque);
	MC_BR_CyclicRead_1.DataType		:= ncPAR_TYP_REAL;
	MC_BR_CyclicRead_1.Mode			:= mcEVERY_RECORD;
	MC_BR_CyclicRead_1();

	MC_BR_CyclicRead_2.Axis			:= ADR(gAxis01);
	MC_BR_CyclicRead_2.Enable		:= TRUE;
	MC_BR_CyclicRead_2.ParID		:= ACP10PAR_PCTRL_S_ACT;
	MC_BR_CyclicRead_2.DataAddress	:= ADR(Axis1EncoderPosition);
	MC_BR_CyclicRead_2.DataType		:= ncPAR_TYP_DINT;
	MC_BR_CyclicRead_2.Mode			:= mcEVERY_RECORD;
	MC_BR_CyclicRead_2();

END_ACTION

ACTION Axis1Param :
	BasicControl.Parameter.Acceleration	:= AutoSequence.par.acceleration;
	BasicControl.Parameter.Deceleration	:= AutoSequence.par.deceleration;
	BasicControl.Parameter.Direction	:= AutoSequence.par.direction[1];
	BasicControl.Parameter.Velocity		:= AutoSequence.par.speedMovement;
	BasicControl.Parameter.Distance		:= AutoSequence.par.distance[1];
	BasicControl.Parameter.HomePosition	:= AutoSequence.par.homePosition[1];
	BasicControl.Parameter.HomeMode		:= AutoSequence.par.homeMode;
	BasicControl.Parameter.Position		:= AutoSequence.par.position[1];

END_ACTION

ACTION Axis1Cmd :
	BasicControl.Command.Power				:= AutoSequence.cmd.powerMotor;
	BasicControl.Command.Home				:= AutoSequence.cmd.home;
	BasicControl.Command.MoveAbsolute		:= AutoSequence.cmd.moveAbsolute[1];
	BasicControl.Command.MoveAdditive		:= AutoSequence.cmd.moveRelative[1];
	BasicControl.Command.Stop				:= AutoSequence.cmd.stopMotor;
	BasicControl.Command.ErrorAcknowledge	:= AutoSequence.cmd.ErrorAcknowledge[1];
END_ACTION
```

### Program Logical/Sources/MotionControl/BasicAxis2 (IEC) - Basic logical control
